// TIA Portal project "Paletizace trayů" (V14)

(* hardware
DEVICE "ET 200S station_1"  ET 200S station
   slot 0: "Rack_0"  Rail
   slot 2: "PLC_1"  IM 151-8 PN/DP CPU  6ES7 151-8AB01-0AB0  V3.2
      slot 1: "PROFINET interface_1"  PN-IO
         slot 1: "Port_1"  Port
         slot 2: "Port_2"  Port
         slot 3: "Port_3"  Port
   slot 4: "PM-E 24VDC_1"  PM-E 24VDC  6ES7 138-4CA01-0AA0
   slot 5: "4SI IO link_1"  4SI IO link  6ES7 138-4GA50-0AB0
   slot 6: "4SI IO link_2"  4SI IO link  6ES7 138-4GA50-0AB0
   slot 7: "4SI IO link_3"  4SI IO link  6ES7 138-4GA50-0AB0
   slot 8: "4SI IO link_4"  4SI IO link  6ES7 138-4GA50-0AB0
   slot 9: "PM-E 24VDC_2"  PM-E 24VDC  6ES7 138-4CA01-0AA0
   slot 10: "8DI x 24VDC_1"  8DI x 24VDC  6ES7 131-4BF00-0AA0
   slot 11: "8DI x 24VDC_2"  8DI x 24VDC  6ES7 131-4BF00-0AA0
   slot 12: "8DI x 24VDC_3"  8DI x 24VDC  6ES7 131-4BF00-0AA0
   slot 13: "8DI x 24VDC_4"  8DI x 24VDC  6ES7 131-4BF00-0AA0
   slot 14: "8DI x 24VDC_5"  8DI x 24VDC  6ES7 131-4BF00-0AA0
   slot 15: "8DI x 24VDC_6"  8DI x 24VDC  6ES7 131-4BF00-0AA0
   slot 16: "8DI x 24VDC_7"  8DI x 24VDC  6ES7 131-4BF00-0AA0
   slot 17: "8DI x 24VDC_8"  8DI x 24VDC  6ES7 131-4BF00-0AA0
   slot 18: "8DI x 24VDC_9"  8DI x 24VDC  6ES7 131-4BF00-0AA0
   slot 19: "8DI x 24VDC_10"  8DI x 24VDC  6ES7 131-4BF00-0AA0
   slot 20: "8DI x 24VDC_11"  8DI x 24VDC  6ES7 131-4BF00-0AA0
   slot 21: "8DI x 24VDC_12"  8DI x 24VDC  6ES7 131-4BF00-0AA0
   slot 22: "8DI x 24VDC_13"  8DI x 24VDC  6ES7 131-4BF00-0AA0
   slot 23: "8DI x 24VDC_14"  8DI x 24VDC  6ES7 131-4BF00-0AA0
   slot 24: "8DI x 24VDC_15"  8DI x 24VDC  6ES7 131-4BF00-0AA0
   slot 25: "8DI x 24VDC_16"  8DI x 24VDC  6ES7 131-4BF00-0AA0
   slot 26: "PM-E 24VDC_3"  PM-E 24VDC  6ES7 138-4CA01-0AA0
   slot 27: "8DO x 24VDC / 0.5A_1"  8DO x 24VDC / 0.5A  6ES7 132-4BF00-0AA0
   slot 28: "8DO x 24VDC / 0.5A_2"  8DO x 24VDC / 0.5A  6ES7 132-4BF00-0AA0
   slot 29: "PM-E 24VDC_4"  PM-E 24VDC  6ES7 138-4CA01-0AA0
   slot 30: "8DO x 24VDC / 0.5A_3"  8DO x 24VDC / 0.5A  6ES7 132-4BF00-0AA0
   slot 31: "8DO x 24VDC / 0.5A_4"  8DO x 24VDC / 0.5A  6ES7 132-4BF00-0AA0
   slot 32: "8DO x 24VDC / 0.5A_5"  8DO x 24VDC / 0.5A  6ES7 132-4BF00-0AA0
   slot 33: "8DO x 24VDC / 0.5A_6"  8DO x 24VDC / 0.5A  6ES7 132-4BF00-0AA0
   slot 34: "8DO x 24VDC / 0.5A_7"  8DO x 24VDC / 0.5A  6ES7 132-4BF00-0AA0
   slot 35: "8DO x 24VDC / 0.5A_8"  8DO x 24VDC / 0.5A  6ES7 132-4BF00-0AA0
   slot 36: "8DO x 24VDC / 0.5A_9"  8DO x 24VDC / 0.5A  6ES7 132-4BF00-0AA0
   slot 37: "8DO x 24VDC / 0.5A_10"  8DO x 24VDC / 0.5A  6ES7 132-4BF00-0AA0
   slot 38: "8DO x 24VDC / 0.5A_11"  8DO x 24VDC / 0.5A  6ES7 132-4BF00-0AA0
   slot 39: "PM-E 24VDC_5"  PM-E 24VDC  6ES7 138-4CA01-0AA0
   slot 40: "8DO x 24VDC / 0.5A_12"  8DO x 24VDC / 0.5A  6ES7 132-4BF00-0AA0
   slot 41: "8DO x 24VDC / 0.5A_13"  8DO x 24VDC / 0.5A  6ES7 132-4BF00-0AA0
   slot 42: "8DO x 24VDC / 0.5A_14"  8DO x 24VDC / 0.5A  6ES7 132-4BF00-0AA0
   slot 43: "8DO x 24VDC / 0.5A_15"  8DO x 24VDC / 0.5A  6ES7 132-4BF00-0AA0
   slot 44: "8DO x 24VDC / 0.5A_16"  8DO x 24VDC / 0.5A  6ES7 132-4BF00-0AA0
   slot 45: "8DO x 24VDC / 0.5A_17"  8DO x 24VDC / 0.5A  6ES7 132-4BF00-0AA0
   slot 46: "8DO x 24VDC / 0.5A_18"  8DO x 24VDC / 0.5A  6ES7 132-4BF00-0AA0
   slot 47: "8DO x 24VDC / 0.5A_19"  8DO x 24VDC / 0.5A  6ES7 132-4BF00-0AA0
   slot 48: "8DO x 24VDC / 0.5A_20"  8DO x 24VDC / 0.5A  6ES7 132-4BF00-0AA0
DEVICE "GSD device_1"  GSD.Device.PN
   slot 0: "Rack"  Rack  V1.0
   slot 0: "ComauR1"  X20IF10E3-1  X20IF10E3-1  2.1.x
      slot 0: "DIM 1"  DIM 1
      slot 1: "Interface"  Interface
         slot 1: "Interface - Port1"  Interface - Port1
         slot 2: "Interface - Port2"  Interface - Port2
   slot 1: "32 Bytes In_1"  32 Bytes In
      slot 0: "17"  17
   slot 2: "32 Bytes Out_1"  32 Bytes Out
      slot 0: "18"  18
DEVICE "GSD device_2"  GSD.Device.PN
   slot 0: "Rack"  Rack  V1.0
   slot 0: "ComauR2"  X20IF10E3-1  X20IF10E3-1  2.1.x
      slot 0: "DIM 1"  DIM 1
      slot 1: "Interface"  Interface
         slot 1: "Interface - Port1"  Interface - Port1
         slot 2: "Interface - Port2"  Interface - Port2
   slot 1: "32 Bytes In_1"  32 Bytes In
      slot 0: "17"  17
   slot 2: "32 Bytes Out_1"  32 Bytes Out
      slot 0: "18"  18
DEVICE "Panel paletizace trayů"  KTP600 Basic color PN
   slot 0: "KTP600 Basic color PN"  KTP600 Basic color PN  6AV6 647-0AD11-3AX0  12.0.0.0
   slot 1: "HMI_RT_2"  KTP600 Basic color PN  6AV6 647-0AD11-3AX0  12.0.0.0
   slot 5: "Panel paletizace trayů.IE_CP_1"  PROFINET Interface  12.0.0.0
      slot 1: "PROFINET Interface_1"  PROFINET Interface
         slot 1: "Port_1"  Port
DEVICE "GSD device_3"  GSD.Device.PN
   slot 0: "Rack"  Rack  V1.0
   slot 1: "rpt1ezp810-8"  plcEZP810-8  6ES7 214-1AG40-0XB0  V4.1
      slot 0: "MasterQ"  MasterQ
      slot 1: "MasterI"  MasterI
      slot 2: "Interface"  Interface
         slot 1: "Port 1"  Port 1
*)

// ===== PLC "PLC_1"  IM 151-8 PN/DP CPU =====

VAR_GLOBAL   // PLC tag table "Default tag table"
   "P12 nahoře" AT %I44.0 : Bool;
   "Zdvih P12B Nahoru" AT %Q17.6 : Bool;
   "Zdvih P12B Brzda" AT %Q18.0 : Bool;
   "Tag_5" AT %M2.0 : Bool;
   "P12 dole" AT %I44.1 : Bool;
   "Zdvih P11B Nahoru" AT %Q17.1 : Bool;
   "Zdvih P12B Dolu" AT %Q17.7 : Bool;
   "Tag_10" AT %Q33.0 : Bool;
   "Tlačítko zapnout" AT %I13.0 : Bool;
   "Tlačítko reset" AT %I13.1 : Bool;
   "Tag_13" AT %Q26.0 : Bool;
   "Tag_14" AT %Q26.1 : Bool;
   "Tag_15" AT %Q26.2 : Bool;
   "FM P35 Start" AT %Q20.3 : Bool;
   "Tag_17" AT %M4.0 : Bool;
   "Reset frekvenčních měničů" AT %Q25.5 : Bool;
   "Tag_19" AT %M4.1 : Bool;
   "Tlačítko override" AT %I13.2 : Bool;
   "Tag_21" AT %M5.0 : Bool;
   "FM P35 rychlost bit 0" AT %Q20.5 : Bool;
   "Tag_12" AT %M6.0 : Bool;
   "FM P35 rychlost bit 1" AT %Q20.6 : Bool;
   "Tag_16" AT %M9.0 : Bool;
   "FM P27 start" AT %Q19.4 : Bool;
   "Tag_20" AT %M4.2 : Bool;
   "Tag_22" AT %M60.0 : Bool;
   "Destohovač P6 nahoru" AT %Q16.3 : Bool;
   "Tag_23" AT %M60.1 : Bool;
   "Destohovač P6 dolu" AT %Q16.4 : Bool;
   "Destohovač P6 brzda" AT %Q16.5 : Bool;
   "Destohovač D6 Nahoře" AT %I40.5 : Bool;
   "Destohovač D6 Dole" AT %I40.7 : Bool;
   "Tag_26" AT %M1.4 : Bool;
   "Dopravník P4 Start" AT %Q16.1 : Bool;
   "Dopravník P5 Stohovač Start" AT %Q16.2 : Bool;
   "Tag_27" AT %M80.1 : Bool;
   "Tag_28" AT %M80.2 : Bool;
   "Dopravník P8 Start" AT %Q16.6 : Bool;
   "Tag_4" AT %M80.4 : Bool;
   "Tag_3" AT %M80.5 : Bool;
   "Dopravník 12 A start" AT %Q17.4 : Bool;
   "Tag_29" AT %M80.6 : Bool;
   "Dopravník 12 A vzad" AT %Q17.5 : Bool;
   "Tag_9" AT %M91.0 : Bool;
   "Dopravník P17 Start" AT %Q18.1 : Bool;
   "Dopravník P18 Start" AT %Q18.2 : Bool;
   "Dopravník Ovinovačka P19 start" AT %Q18.3 : Bool;
   "Tag_30" AT %M91.1 : Bool;
   "Tag_31" AT %M91.2 : Bool;
   "Tag_32" AT %M91.3 : Bool;
   "Dopravník P20 Start" AT %Q18.4 : Bool;
   "Tag_33" AT %M20.0 : Bool;
   "Tag_34" AT %M20.1 : Bool;
   "Zdvih P11B Dolu" AT %Q17.2 : Bool;
   "Zdvih P11B Brzda" AT %Q17.3 : Bool;
   "P11 dole" AT %I42.7 : Bool;
   "P11 nahoře" AT %I42.6 : Bool;
   "Tag_8" AT %M20.2 : Bool;
   "Dopravník P11A start" AT %Q16.7 : Bool;
   "Dopravník P11A vzad" AT %Q17.0 : Bool;
   "Tag_39" AT %M20.4 : Bool;
   "Tag_35" AT %M110.0 : Bool;
   "Dopravník P36 start" AT %Q20.7 : Bool;
   "Dopravník P37 Start" AT %Q21.0 : Bool;
   "Tag_36" AT %M110.1 : Bool;
   "FM P23.1 Start" AT %Q186.1 : Bool;
   "FM P23.2 Start" AT %Q19.1 : Bool;
   "FM P28 Start" AT %Q20.0 : Bool;
   "FM P29 Start" AT %Q20.1 : Bool;
   "P33 Start" AT %Q20.2 : Bool;
   "Tag_18" AT %Q19.6 : Bool;
   "Tag_40" AT %Q19.7 : Bool;
   "P 47.1 Start" AT %Q21.2 : Bool;
   "P 47.2 Start" AT %Q21.3 : Bool;
   "P 49 Start" AT %Q21.4 : Bool;
   "Rovnání palety P12 sevřít" AT %Q47.5 : Bool;
   "Rovnání palety P12 rozevřít" AT %Q47.4 : Bool;
   "Rovnání palety P11 sevřít" AT %Q47.1 : Bool;
   "Rovnání palety P11 rozevřít" AT %Q47.0 : Bool;
   "Destohovač sevřít" AT %Q41.7 : Bool;
   "Destohovač rozevřít" AT %Q41.6 : Bool;
   "Klapka 47.2 nahoru" AT %Q46.2 : Bool;
   "Klapka 47.2 dolů" AT %Q46.3 : Bool;
   "Klapka P47.1 nahoru" AT %Q46.0 : Bool;
   "Klapka P47.1 dolů" AT %Q46.1 : Bool;
   "Klapka P33 nahoru" AT %Q46.4 : Bool;
   "Klapka P33 dolů" AT %Q46.5 : Bool;
   "Paleta na konci P5" AT %I41.4 : Bool;
   "Destohovač D6 rameno pravé sevřeno" AT %I41.3 : Bool;
   "Paleta na P8 pozice 12" AT %I42.3 : Bool;
   "Tag_1" AT %I44.5 : Bool;
   "Paleta na P12" AT %I44.2 : Bool;
   "Tag_7" AT %Q47.2 : Bool;
   "PaletaNaD17pozice12" AT %I44.6 : Bool;
   "Tag_41" AT %T50 : Timer;
   "Paleta na konci P17" AT %I48.0 : Bool;
   "Tag_42" AT %T51 : Timer;
   "Spoždění ukončení automatu" AT %T0 : Timer;
   "Paleta na konci P18" AT %I48.1 : Bool;
   "Paleta v ovíječce P19" AT %I48.2 : Bool;
   "Paleta na Začátku P18" AT %I48.7 : Bool;
   "Paleta na Začátku P20" AT %I48.4 : Bool;
   "Paleta na konci P20" AT %I48.5 : Bool;
   "Karton na konci P47.2" AT %I55.1 : Bool;
   "Karton na začátku P49" AT %I59.1 : Bool;
   "Tag_43" AT %T40 : Timer;
   "Karton na konci P49" AT %I58.6 : Bool;
   "Konec řady na P49" AT %I58.7 : Bool;
   "Dojetá řada na P49" AT %I59.0 : Bool;
   "Karton na konci P47.1" AT %I55.2 : Bool;
   "Dopravník P47.2 plný" AT %I45.5 : Bool;
   "Tag_44" AT %M10.0 : Bool;
   "Tag_45" AT %M11.0 : Bool;
   "Tag_46" AT %M16.0 : Bool;
   "Tag_47" AT %M16.1 : Bool;
   "Tag_48" AT %T60 : Timer;
   "Tag_49" AT %T61 : Timer;
   "Tag_50" AT %T62 : Timer;
   "Tag_51" AT %T63 : Timer;
   "Silové obvody okruh 1 OK" AT %I14.0 : Bool;
   "Motorový jistič Destohovač D6 OK" AT %I0.1 : Bool;
   "Destohovač D6 havárie dole" AT %I0.7 : Bool;
   "Destohovač D6 havárie nahoře" AT %I0.6 : Bool;
   "Tlak vzduchu OK" AT %I3.7 : Bool;
   "Paleta pod destohovačem D6" AT %I40.4 : Bool;
   "Destohovač D6 Uprostřed" AT %I40.6 : Bool;
   "Destohovač D6 Rameno Levé otevřeno" AT %I41.0 : Bool;
   "Destohovač D6 rameno pravé otevřeno" AT %I41.2 : Bool;
   "Destohovač D6 rameno levé sevřeno" AT %I41.1 : Bool;
   "Tag_62" AT %I320.0 : Bool;
   "Tag_63" AT %M150.0 : Bool;
   "Tag_64" AT %M150.3 : Bool;
   "Tag_65" AT %Q320.0 : Bool;
   "Tag_66" AT %M100.0 : Bool;
   "Tag_67" AT %M100.1 : Bool;
   "Tag_68" AT %M120.0 : Bool;
   "Motorový jistič P3,P4,P5,P8 OK" AT %I0.0 : Bool;
   "Paleta na Začátku D8" AT %I45.6 : Bool;
   "Stoh palet na konci D4" AT %I40.2 : Bool;
   "Stoh palet na Začátku D5" AT %I40.3 : Bool;
   "Paleta na P8 pozice 11" AT %I42.2 : Bool;
   "Pomocná začátek přesunu na D12" AT %M61.1 : Bool;
   "Tag_24" AT %M120.1 : Bool;
   "Starttovací okno D18" AT %T52 : Timer;
   "Tag_25" AT %T41 : Timer;
   "Tag_37" AT %I54.7 : Bool;
   "Tag_38" AT %I54.3 : Bool;
   "Tag_52" AT %I54.1 : Bool;
   "Tag_53" AT %I54.4 : Bool;
   "Tag_54" AT %T42 : Timer;
   "Tag_55" AT %T44 : Timer;
   "Tag_56" AT %I54.2 : Bool;
   "Tag_57" AT %I54.0 : Bool;
   "Tag_58" AT %T45 : Timer;
   "Tag_59" AT %Q33.1 : Bool;
   "Tag_60" AT %Q33.3 : Bool;
   "Tag_70" AT %Q33.4 : Bool;
   "Tag_71" AT %Q33.5 : Bool;
   "Tag_72" AT %M2.1 : Bool;
   "Tag_73" AT %M2.2 : Bool;
   "Tag_2" AT %T2 : Timer;
   "Tag_6" AT %T90 : Timer;
   "Tag_11" AT %T91 : Timer;
END_VAR

VAR_GLOBAL   // PLC tag table "Tag table_1"
   "Ovíječka_Volná trať" AT %I10.0 : Bool;
   "Ovíječka_Konec balení" AT %I10.1 : Bool;
   "Ovíječka_Porucha" AT %I10.2 : Bool;
   "Ovíječka_Paleta na točně" AT %I10.3 : Bool;
   "Ovíječce_Start balení" AT %Q29.4 : Bool;
   "Ovíječce_Možno balit" AT %Q29.5 : Bool;
   "Tag_61" AT %Q29.6 : Bool;
   "Tag_69" AT %Q29.7 : Bool;
END_VAR

VAR_GLOBAL   // PLC tag table "System"
   "AlwaysTRUE" AT %M1.2 : Bool;
   "Clock memory bit 10 Hz" AT %M0.0 : Bool;
   "Clock memory bit 5 Hz" AT %M0.1 : Bool;
   "Clock memory bit 2.5 Hz" AT %M0.2 : Bool;
   "Clock memory bit 2 Hz" AT %M0.3 : Bool;
   "Clock memory bit 1.25 Hz" AT %M0.4 : Bool;
   "Clock memory bit 1 Hz" AT %M0.5 : Bool;
   "Clock memory bit 0.625 Hz" AT %M0.6 : Bool;
   "Clock memory bit 0.5 Hz" AT %M0.7 : Bool;
   "AlwaysFALSE" AT %M1.3 : Bool;
   "DiagStatusUpdate" AT %M1.1 : Bool;
   "FirstScan" AT %M1.0 : Bool;
END_VAR

TYPE "Artikl2"
   STRUCT
      Cislo : Int;
      Pocet : Int;
      Novy : Bool;
      Mlecny : Bool;
   END_STRUCT;
END_TYPE

TYPE "Artikl"
   STRUCT
      Novy : Bool;
      Mlecny : Bool;
      Mlecny4 : Bool;
      Mlecny6 : Bool;
      Mlecny8 : Bool;
      Mlecny9 : Bool;
      Mlecny99 : Bool;
      Mlecny9999 : Bool;
      Cislo : Word;
      Pocet : Word;
   END_STRUCT;
END_TYPE

TYPE "Pocet"
   STRUCT
      "Požadovaný počet vrstev" : Int;
      "Aktuální počet vrstev" : Int;
      "Aktuální počet půlvrstev" : Int;
   END_STRUCT;
END_TYPE

TYPE "Paleta"
   STRUCT
      Artik : String;
      "Počet vrstev" : Int;
      "Počet půlvrstev" : Int;
      "Neúplná paleta" : Bool;
   END_STRUCT;
END_TYPE

DATA_BLOCK "OB1"   // DB1
{ S7_Optimized_Access := 'FALSE' }
VERSION : 0.1
   VAR
      OB1_EV_CLASS : Byte;
      OB1_SCAN_1 : Byte;
      OB1_PRIORITY : Byte;
      OB1_OB_NUMBR : Byte;
      OB1_RESERVED_1 : Byte;
      OB1_RESERVED_2 : Byte;
      OB1_PREV_CYCLE : Int;
      OB1_MIN_CYCLE : Int;
      OB1_MAX_CYCLE : Int;
      OB1_DATE_TIME : Date_And_Time;
   END_VAR
BEGIN
END_DATA_BLOCK

DATA_BLOCK "Data_block_1"   // DB2
{ S7_Optimized_Access := 'FALSE' }
VERSION : 0.1
   VAR
      moje : Struct
         aa : Bool;
         aaaa : Bool;
      END_STRUCT;
      dd : Bool;
   END_VAR
BEGIN
END_DATA_BLOCK

DATA_BLOCK "Data_block_2"   // DB3
{ S7_Optimized_Access := 'FALSE' }
VERSION : 0.1
BEGIN
END_DATA_BLOCK

DATA_BLOCK "DataPole"   // DB4
{ S7_Optimized_Access := 'FALSE' }
VERSION : 0.1
   VAR
      Artikly : Array[0..100] of "Artikl2";
      Konci : Bool;
   END_VAR
BEGIN
END_DATA_BLOCK

DATA_BLOCK "Block_1_DB"   // DB5
{ S7_Optimized_Access := 'FALSE' }
VERSION : 0.1
// stored: InstanceOfName Block_1
"Block_1"
BEGIN
END_DATA_BLOCK

DATA_BLOCK "ArtiklDB"   // DB6
{ S7_Optimized_Access := 'FALSE' }
VERSION : 0.1
   VAR
      Artikl : "Artikl";
   END_VAR
BEGIN
END_DATA_BLOCK

DATA_BLOCK "Dopravníky palet_DB"   // DB8
{ S7_Optimized_Access := 'FALSE' }
VERSION : 0.1
// stored: InstanceOfName Dopravníky palet
"Dopravníky palet"
BEGIN
END_DATA_BLOCK

DATA_BLOCK "Data_block_3"   // DB9
{ S7_Optimized_Access := 'FALSE' }
VERSION : 0.1
   VAR
      artikl : Struct
         Novy : Bool;
         Mlecny : Bool;
         Mlecny4 : Bool;
         Mlecny6 : Bool;
         Mlecny8 : Bool;
         Mlecny9 : Bool;
         Mlecny99 : Bool;
         Mlecny9999 : Bool;
         Cislo : Word;
         Pocet : Word;
      END_STRUCT;
   END_VAR
BEGIN
END_DATA_BLOCK

DATA_BLOCK "Artikly"   // DB10
{ S7_Optimized_Access := 'FALSE' }
VERSION : 0.1
   VAR
      Artikly : Array[0..100] of "Artikl";
   END_VAR
BEGIN
END_DATA_BLOCK

DATA_BLOCK "Dopravníky kartonů linka 1_DB"   // DB11
{ S7_Optimized_Access := 'FALSE' }
VERSION : 0.1
// stored: InstanceOfName Dopravníky kartonů linka 1
"Dopravníky kartonů linka 1"
BEGIN
END_DATA_BLOCK

DATA_BLOCK "Globální řízení_DB"   // DB12
{ S7_Optimized_Access := 'FALSE' }
VERSION : 0.1
// stored: InstanceOfName Globální řízení
"Globální řízení"
BEGIN
END_DATA_BLOCK

DATA_BLOCK "Počítadlo_DB"   // DB15
{ S7_Optimized_Access := 'FALSE' }
VERSION : 0.1
// stored: InstanceOfName Počítadlo
"Počítadlo"
BEGIN
END_DATA_BLOCK

DATA_BLOCK "OPPovely"   // DB20
{ S7_Optimized_Access := 'FALSE' }
VERSION : 0.1
   VAR
      "OP Start" : Bool;
      "OP Stop" : Bool;
      "OP Manual" : Bool;
      "P3 Start" : Bool;
      "P4 Start" : Bool;
      "P5 Start" : Bool;
      "Destohovač nahoru" : Bool;
      "Destohovač dolu" : Bool;
      "Destohovač ramena sevřít" : Bool;
      "Destohovač ramena rozevřít" : Bool;
      "P8 Start" : Bool;
      "P12 Start" : Bool;
      "P12 Vzad" : Bool;
      "P12 Nahoru" : Bool;
      "P12 Dolu" : Bool;
      "P12 Rovnání" : Bool;
      "P11 Start" : Bool;
      "P11 Vzad" : Bool;
      "P11 Nahoru" : Bool;
      "P11 Dolu" : Bool;
      "P11 Rovnání" : Bool;
      "P17 Start" : Bool;
      "P18 Start" : Bool;
      "P19 Ovíječka Start" : Bool;
      "P20 Start" : Bool;
      "P21 Start" : Bool;
      Linka1 : Struct
         "P23 Start" : Bool;
         "P28 Start" : Bool;
         "P27 Elevátor Start" : Bool;
         "P29 Start" : Bool;
         "P33 Start" : Bool;
         "Klapka P33" : Bool;
         "P36 Start" : Bool;
         "P35 Elevátor Start" : Bool;
         "P37 Start" : Bool;
         "P47.1 Start" : Bool;
         "Klapka P47.1" : Bool;
         "P47.2 Start" : Bool;
         "Klapka P47.2" : Bool;
         "P49 Start" : Bool;
         reserve : Word;
      END_STRUCT;
   END_VAR
BEGIN
END_DATA_BLOCK

DATA_BLOCK "OPPovely Positivní Hrana"   // DB21
{ S7_Optimized_Access := 'FALSE' }
VERSION : 0.1
   VAR
      "OP Start" : Bool;
      "OP Stop" : Bool;
      "OP Manual" : Bool;
      "P3 Start" : Bool;
      "P4 Start" : Bool;
      "P5 Start" : Bool;
      "Destohovač nahoru" : Bool;
      "Destohovač dolu" : Bool;
      "Destohovač ramena sevřít" : Bool;
      "Destohovač ramena rozevřít" : Bool;
      "P8 Start" : Bool;
      "P12 Start" : Bool;
      "P12 Vzad" : Bool;
      "P12 Nahoru" : Bool;
      "P12 Dolu" : Bool;
      "P12 Rovnání" : Bool;
      "P11 Start" : Bool;
      "P11 Vzad" : Bool;
      "P11 Nahoru" : Bool;
      "P11 Dolu" : Bool;
      "P11 Rovnání" : Bool;
      "P17 Start" : Bool;
      "P18 Start" : Bool;
      "P19 Ovíječka Start" : Bool;
      "P20 Start" : Bool;
      "P21 Start" : Bool;
      Linka1 : Struct
         "P23 Start" : Bool;
         "P28 Start" : Bool;
         "P27 Elevátor Start" : Bool;
         "P29 Start" : Bool;
         "P33 Start" : Bool;
         "Klapka P33" : Bool;
         "P36 Start" : Bool;
         "P35 Elevátor Start" : Bool;
         "P37 Start" : Bool;
         "P47.1 Start" : Bool;
         "Klapka P47.1" : Bool;
         "P47.2 Start" : Bool;
         "Klapka P47.2" : Bool;
         "P49 Start" : Bool;
         reserve : Word;
      END_STRUCT;
   END_VAR
BEGIN
END_DATA_BLOCK

DATA_BLOCK "OPPovely Negativní Hrana"   // DB22
{ S7_Optimized_Access := 'FALSE' }
VERSION : 0.1
   VAR
      "OP Start" : Bool;
      "OP Stop" : Bool;
      "OP Manual" : Bool;
      "P3 Start" : Bool;
      "P4 Start" : Bool;
      "P5 Start" : Bool;
      "Destohovač nahoru" : Bool;
      "Destohovač dolu" : Bool;
      "Destohovač ramena sevřít" : Bool;
      "Destohovač ramena rozevřít" : Bool;
      "P8 Start" : Bool;
      "P12 Start" : Bool;
      "P12 Vzad" : Bool;
      "P12 Nahoru" : Bool;
      "P12 Dolu" : Bool;
      "P12 Rovnání" : Bool;
      "P11 Start" : Bool;
      "P11 Vzad" : Bool;
      "P11 Nahoru" : Bool;
      "P11 Dolu" : Bool;
      "P11 Rovnání" : Bool;
      "P17 Start" : Bool;
      "P18 Start" : Bool;
      "P19 Ovíječka Start" : Bool;
      "P20 Start" : Bool;
      "P21 Start" : Bool;
      Linka1 : Struct
         "P23 Start" : Bool;
         "P28 Start" : Bool;
         "P27 Elevátor Start" : Bool;
         "P29 Start" : Bool;
         "P33 Start" : Bool;
         "Klapka P33" : Bool;
         "P36 Start" : Bool;
         "P35 Elevátor Start" : Bool;
         "P37 Start" : Bool;
         "P47.1 Start" : Bool;
         "Klapka P47.1" : Bool;
         "P47.2 Start" : Bool;
         "Klapka P47.2" : Bool;
         "P49 Start" : Bool;
         reserve : Word;
      END_STRUCT;
   END_VAR
BEGIN
END_DATA_BLOCK

FUNCTION_BLOCK "Block_1"   // FB1, LAD
{ S7_Optimized_Access := 'FALSE' }
VERSION : 0.1
BEGIN
END_FUNCTION_BLOCK

FUNCTION_BLOCK "Dopravníky palet"   // FB2, LAD
{ S7_Optimized_Access := 'FALSE' }
VERSION : 0.1
   VAR
      Přesun : Struct
         KonecD4naDestohovač : Bool;
         DestohovačNaKonecD5 : Bool;
         KonecD5naZačátekD8 : Bool;
         ZačátekD8naD8x12 : Bool;
         D8x12naD8x11 : Bool;
         D8x12naD12 : Bool;
         D8x11naD11 : Bool;
         D12naD17x12 : Bool;
         D11naD17x11 : Bool;
         D17x12naKonecP17 : Bool;
         D17x11naKonecP17 : Bool;
         KonecP17naZačátekP18 : Bool;
         ZačátekP18naKonecP18 : Bool;
         KonecP18naP19 : Bool;
         P19naZačátekP20 : Bool;
         ZačátekP20naKonecP20 : Bool;
         KonecP20NaP21 : Bool;
      END_STRUCT;
      "Přesun zahájen" : Struct
         KonecD4naDestohovač : Bool;
         DestohovačNaKonecD5 : Bool;
         KonecD5naZačátekD8 : Bool;
         ZačátekD8naD8x12 : Bool;
         D8x12naD8x11 : Bool;
         D8x12naD12 : Bool;
         D8x11naD11 : Bool;
         D12naD17x12 : Bool;
         D11naD17x11 : Bool;
         D17x12naKonecP17 : Bool;
         D17x11naKonecP17 : Bool;
         KonecP17naZačátekP18 : Bool;
         ZačátekP18naKonecP18 : Bool;
         KonecP18naP19 : Bool;
         P19naZačátekP20 : Bool;
         ZačátekP20naKonecP20 : Bool;
         KonecP20NaP21 : Bool;
      END_STRUCT;
      "Přesun zahájen paměť hrany" : Struct
         KonecD4naDestohovač : Bool;
         DestohovačNaKonecD5 : Bool;
         KonecD5naZačátekD8 : Bool;
         ZačátekD8naD8x12 : Bool;
         D8pozice12naD8x11 : Bool;
         D8x12naD12 : Bool;
         D8x11naD11 : Bool;
         D12naD17x12 : Bool;
         D11naD17x11 : Bool;
         D17x12naKonecP17 : Bool;
         D17x11naKonecP17 : Bool;
         KonecP17naZačátekP18 : Bool;
         ZačátekP18naKonecP18 : Bool;
         KonecP18naP19 : Bool;
         P19naZačátekP20 : Bool;
         ZačátekP20naKonecP20 : Bool;
         KonecP20NaP21 : Bool;
      END_STRUCT;
      "Přítomnosti palet" : Struct
         PaletaPodDestohovačem : Bool;
         PaletaNaKonciD5 : Bool;
         PaletaNaZačátkuD8 : Bool;
         PaletaNaD8pozice12 : Bool;
         PaletaNaD8pozice11 : Bool;
         PaletaNaP12 : Bool;
         PaletaNaP11 : Bool;
         PaletaNaD17pozice12 : Bool;
         PaletaNaD17pozice11 : Bool;
         PaletaNaKonciP17 : Bool;
         "PaletaNaZačátku P18" : Bool;
         PaletaNaKonciP18 : Bool;
         PaletaNaP19 : Bool;
         PaletaNaZačátkuP20 : Bool;
         PaletaNaKonciP20 : Bool;
      END_STRUCT;
      "Nájezdy palet" : Struct
         PaletaPodDestohovačem : Bool;
         PaletaNaKonciD5 : Bool;
         PaletaNaZačátkuD8 : Bool;
         PaletaNaD8pozice12 : Bool;
         PaletaNaD8pozice11 : Bool;
         PaletaNaP12 : Bool;
         PaletaNaP11 : Bool;
         PaletaNaD17pozice12 : Bool;
         PaletaNaD17pozice11 : Bool;
         PaletaNaKonciP17 : Bool;
         "PaletaNaZačátku P18" : Bool;
         PaletaNaKonciP18 : Bool;
         PaletaNaP19 : Bool;
         PaletaNaZačátkuP20 : Bool;
         PaletaNaKonciP20 : Bool;
      END_STRUCT;
      Palety : Struct
         P12 : "Paleta";
         P11 : "Paleta";
         P17poziceP11 : "Paleta";
         P17poziceP12 : "Paleta";
         KonecP17 : "Paleta";
         ZačátekP18 : "Paleta";
         KonecP18 : "Paleta";
         P19 : "Paleta";
         ZačátekP20 : "Paleta";
      END_STRUCT;
      Hrany : Struct
         T51Negativní : Bool;
      END_STRUCT;
      "Pallet dispenser_Instance" : "Pallet dispenser";
      "Přítomnost palety_Instance" : "Přítomnost palety";
   END_VAR
   VAR_TEMP
      Dummy : Bool;
      "Rovnání P11 sevřít" : Bool;
      "Rovnání P11 rozevřít" : Bool;
      "Rovnání P12 sevřít" : Bool;
      "Rovnání P12 rozevřít" : Bool;
      "Destohovač sevřít" : Bool;
      "Destohovač rozevřít" : Bool;
      "D12 Nahoru" : Bool;
   END_VAR
   VAR_TEMP   // added for the SCL form of the ladder/FBD networks
      _s5time1 : S5Time;
      _w1 : Bool;
      _w2 : Bool;
      _w3 : Bool;
   END_VAR
BEGIN

REGION Network 1
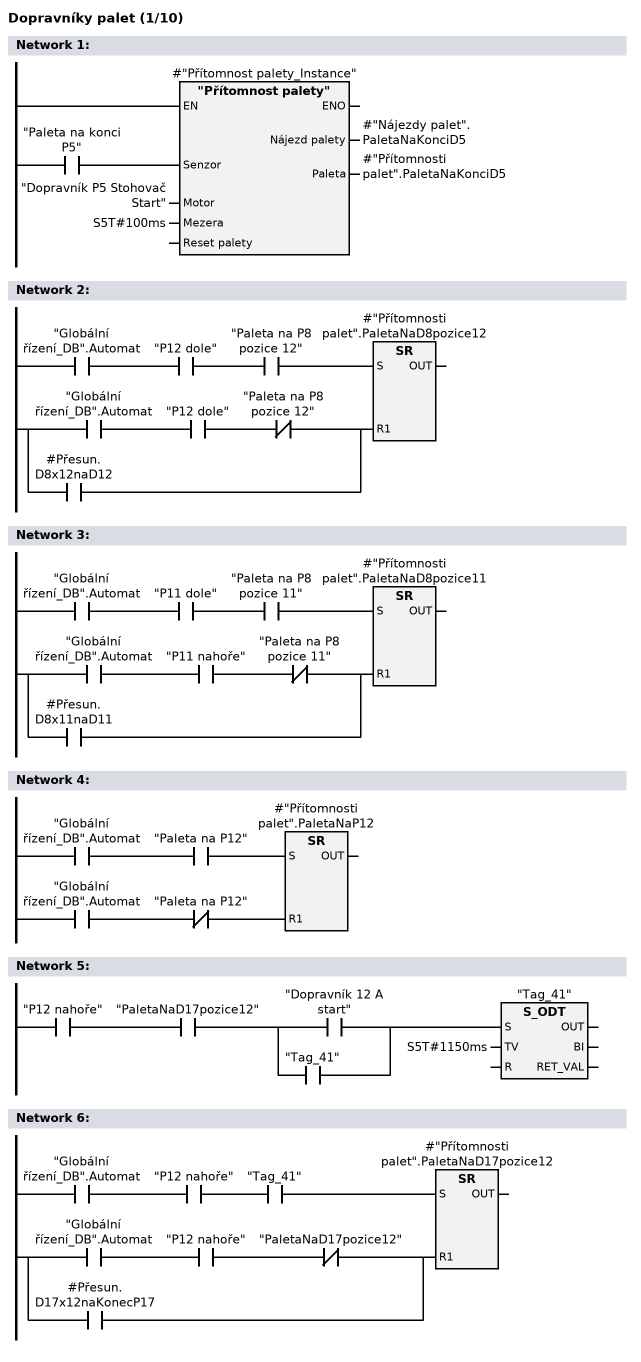
   RUNG wire#powerrail
      #"Přítomnost palety_Instance"(Senzor := wire#w1, Motor := "Dopravník P5 Stohovač Start", Mezera := S5T#100ms, "Reset palety" :=, "Nájezd palety" => #"Nájezdy palet".PaletaNaKonciD5, Paleta => #"Přítomnosti palet".PaletaNaKonciD5)
   END_RUNG
   RUNG wire#powerrail
      Contact( "Paleta na konci P5" )
   END_RUNG wire#w1
   // the same network as SCL:
   #"Přítomnost palety_Instance"(Senzor := "Paleta na konci P5",   // "Přítomnost palety"
                           Motor := "Dopravník P5 Stohovač Start",
                           Mezera := S5T#100ms,
                           "Nájezd palety" => #"Nájezdy palet".PaletaNaKonciD5,
                           Paleta => #"Přítomnosti palet".PaletaNaKonciD5);
END_REGION

REGION Network 2
   RUNG wire#powerrail
      Contact( "Globální řízení_DB".Automat )
      Contact( "P12 dole" )
      Contact( "Paleta na P8 pozice 12" )
      S_SR(operand := #"Přítomnosti palet".PaletaNaD8pozice12, r1 := wire#w1)
   END_RUNG
   RUNG wire#powerrail
      Contact( "Globální řízení_DB".Automat )
      Contact( "P12 dole" )
      I_Contact( "Paleta na P8 pozice 12" )
   END_RUNG wire#w1
   RUNG wire#powerrail
      Contact( #Přesun.D8x12naD12 )
   END_RUNG wire#w1
   // the same network as SCL:
   IF "Globální řízení_DB".Automat AND "P12 dole" AND "Paleta na P8 pozice 12" THEN
       #"Přítomnosti palet".PaletaNaD8pozice12 := TRUE;   // SR flip-flop
   END_IF;
   IF ("Globální řízení_DB".Automat AND "P12 dole" AND NOT "Paleta na P8 pozice 12") OR #Přesun.D8x12naD12 THEN
       #"Přítomnosti palet".PaletaNaD8pozice12 := FALSE;
   END_IF;
END_REGION

REGION Network 3
   RUNG wire#powerrail
      Contact( "Globální řízení_DB".Automat )
      Contact( "P11 dole" )
      Contact( "Paleta na P8 pozice 11" )
      S_SR(operand := #"Přítomnosti palet".PaletaNaD8pozice11, r1 := wire#w1)
   END_RUNG
   RUNG wire#powerrail
      Contact( "Globální řízení_DB".Automat )
      Contact( "P11 nahoře" )
      I_Contact( "Paleta na P8 pozice 11" )
   END_RUNG wire#w1
   RUNG wire#powerrail
      Contact( #Přesun.D8x11naD11 )
   END_RUNG wire#w1
   // the same network as SCL:
   IF "Globální řízení_DB".Automat AND "P11 dole" AND "Paleta na P8 pozice 11" THEN
       #"Přítomnosti palet".PaletaNaD8pozice11 := TRUE;   // SR flip-flop
   END_IF;
   IF ("Globální řízení_DB".Automat AND "P11 nahoře" AND NOT "Paleta na P8 pozice 11") OR #Přesun.D8x11naD11 THEN
       #"Přítomnosti palet".PaletaNaD8pozice11 := FALSE;
   END_IF;
END_REGION

REGION Network 4
   RUNG wire#powerrail
      Contact( "Globální řízení_DB".Automat )
      Contact( "Paleta na P12" )
      S_SR(operand := #"Přítomnosti palet".PaletaNaP12, r1 := wire#w1)
   END_RUNG
   RUNG wire#powerrail
      Contact( "Globální řízení_DB".Automat )
      I_Contact( "Paleta na P12" )
   END_RUNG wire#w1
   // the same network as SCL:
   IF "Globální řízení_DB".Automat AND "Paleta na P12" THEN
       #"Přítomnosti palet".PaletaNaP12 := TRUE;   // SR flip-flop
   END_IF;
   IF "Globální řízení_DB".Automat AND NOT "Paleta na P12" THEN
       #"Přítomnosti palet".PaletaNaP12 := FALSE;
   END_IF;
END_REGION

REGION Network 5
   RUNG wire#powerrail
      Contact( "P12 nahoře" )
      Contact( "PaletaNaD17pozice12" )
      wire#w1
      Contact( "Dopravník 12 A start" )
      wire#w2
      S_ODT(T_NO := "Tag_41", TV := S5T#1150ms, R :=, BI =>, RET_VAL =>)
   END_RUNG
   RUNG wire#w1
      Contact( "Tag_41" )
   END_RUNG wire#w2
   // the same network as SCL:
   #_s5time1 := S_ODT(T_NO := "Tag_41",
                      S := "P12 nahoře" AND "PaletaNaD17pozice12" AND ("Dopravník 12 A start" OR "Tag_41"),
                      TV := S5T#1150ms);
END_REGION

REGION Network 6
   RUNG wire#powerrail
      Contact( "Globální řízení_DB".Automat )
      Contact( "P12 nahoře" )
      Contact( "Tag_41" )
      S_SR(operand := #"Přítomnosti palet".PaletaNaD17pozice12, r1 := wire#w1)
   END_RUNG
   RUNG wire#powerrail
      Contact( "Globální řízení_DB".Automat )
      Contact( "P12 nahoře" )
      I_Contact( "PaletaNaD17pozice12" )
   END_RUNG wire#w1
   RUNG wire#powerrail
      Contact( #Přesun.D17x12naKonecP17 )
   END_RUNG wire#w1
   // the same network as SCL:
   IF "Globální řízení_DB".Automat AND "P12 nahoře" AND "Tag_41" THEN
       #"Přítomnosti palet".PaletaNaD17pozice12 := TRUE;   // SR flip-flop
   END_IF;
   IF ("Globální řízení_DB".Automat AND "P12 nahoře" AND NOT "PaletaNaD17pozice12") OR #Přesun.D17x12naKonecP17 THEN
       #"Přítomnosti palet".PaletaNaD17pozice12 := FALSE;
   END_IF;
END_REGION

REGION Network 7
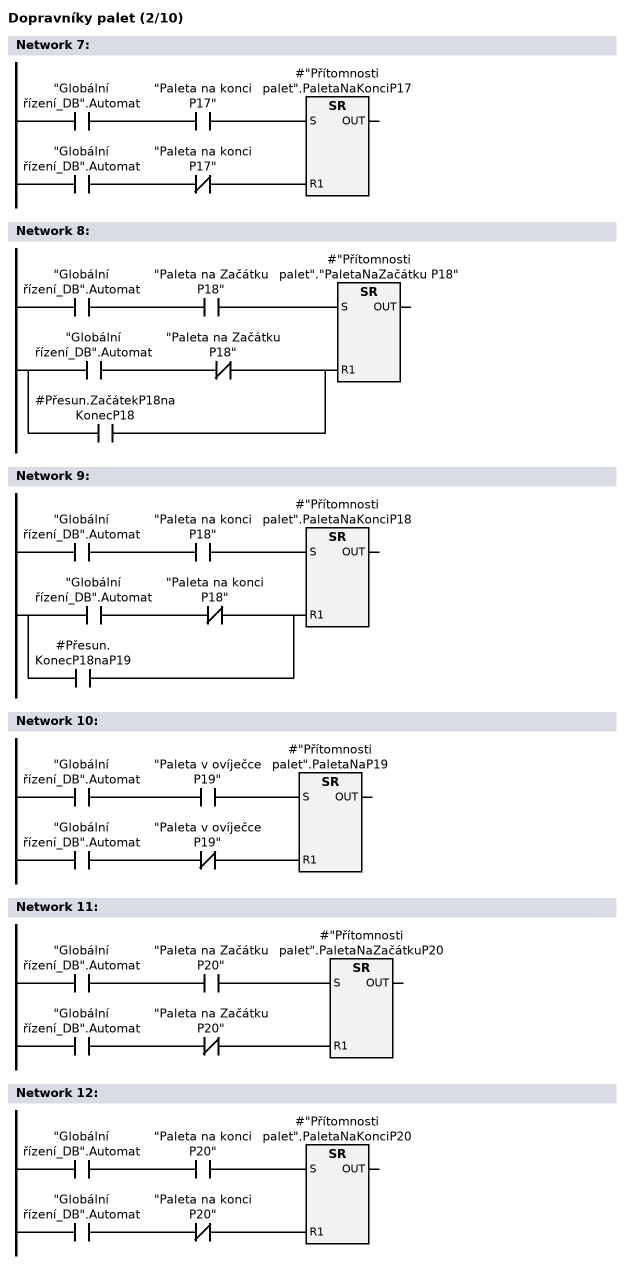
   RUNG wire#powerrail
      Contact( "Globální řízení_DB".Automat )
      Contact( "Paleta na konci P17" )
      S_SR(operand := #"Přítomnosti palet".PaletaNaKonciP17, r1 := wire#w1)
   END_RUNG
   RUNG wire#powerrail
      Contact( "Globální řízení_DB".Automat )
      I_Contact( "Paleta na konci P17" )
   END_RUNG wire#w1
   // the same network as SCL:
   IF "Globální řízení_DB".Automat AND "Paleta na konci P17" THEN
       #"Přítomnosti palet".PaletaNaKonciP17 := TRUE;   // SR flip-flop
   END_IF;
   IF "Globální řízení_DB".Automat AND NOT "Paleta na konci P17" THEN
       #"Přítomnosti palet".PaletaNaKonciP17 := FALSE;
   END_IF;
END_REGION

REGION Network 8
   RUNG wire#powerrail
      Contact( "Globální řízení_DB".Automat )
      Contact( "Paleta na Začátku P18" )
      S_SR(operand := #"Přítomnosti palet"."PaletaNaZačátku P18", r1 := wire#w1)
   END_RUNG
   RUNG wire#powerrail
      Contact( "Globální řízení_DB".Automat )
      I_Contact( "Paleta na Začátku P18" )
   END_RUNG wire#w1
   RUNG wire#powerrail
      Contact( #Přesun.ZačátekP18naKonecP18 )
   END_RUNG wire#w1
   // the same network as SCL:
   IF "Globální řízení_DB".Automat AND "Paleta na Začátku P18" THEN
       #"Přítomnosti palet"."PaletaNaZačátku P18" := TRUE;   // SR flip-flop
   END_IF;
   IF ("Globální řízení_DB".Automat AND NOT "Paleta na Začátku P18") OR #Přesun.ZačátekP18naKonecP18 THEN
       #"Přítomnosti palet"."PaletaNaZačátku P18" := FALSE;
   END_IF;
END_REGION

REGION Network 9
   RUNG wire#powerrail
      Contact( "Globální řízení_DB".Automat )
      Contact( "Paleta na konci P18" )
      S_SR(operand := #"Přítomnosti palet".PaletaNaKonciP18, r1 := wire#w1)
   END_RUNG
   RUNG wire#powerrail
      Contact( "Globální řízení_DB".Automat )
      I_Contact( "Paleta na konci P18" )
   END_RUNG wire#w1
   RUNG wire#powerrail
      Contact( #Přesun.KonecP18naP19 )
   END_RUNG wire#w1
   // the same network as SCL:
   IF "Globální řízení_DB".Automat AND "Paleta na konci P18" THEN
       #"Přítomnosti palet".PaletaNaKonciP18 := TRUE;   // SR flip-flop
   END_IF;
   IF ("Globální řízení_DB".Automat AND NOT "Paleta na konci P18") OR #Přesun.KonecP18naP19 THEN
       #"Přítomnosti palet".PaletaNaKonciP18 := FALSE;
   END_IF;
END_REGION

REGION Network 10
   RUNG wire#powerrail
      Contact( "Globální řízení_DB".Automat )
      Contact( "Paleta v ovíječce P19" )
      S_SR(operand := #"Přítomnosti palet".PaletaNaP19, r1 := wire#w1)
   END_RUNG
   RUNG wire#powerrail
      Contact( "Globální řízení_DB".Automat )
      I_Contact( "Paleta v ovíječce P19" )
   END_RUNG wire#w1
   // the same network as SCL:
   IF "Globální řízení_DB".Automat AND "Paleta v ovíječce P19" THEN
       #"Přítomnosti palet".PaletaNaP19 := TRUE;   // SR flip-flop
   END_IF;
   IF "Globální řízení_DB".Automat AND NOT "Paleta v ovíječce P19" THEN
       #"Přítomnosti palet".PaletaNaP19 := FALSE;
   END_IF;
END_REGION

REGION Network 11
   RUNG wire#powerrail
      Contact( "Globální řízení_DB".Automat )
      Contact( "Paleta na Začátku P20" )
      S_SR(operand := #"Přítomnosti palet".PaletaNaZačátkuP20, r1 := wire#w1)
   END_RUNG
   RUNG wire#powerrail
      Contact( "Globální řízení_DB".Automat )
      I_Contact( "Paleta na Začátku P20" )
   END_RUNG wire#w1
   // the same network as SCL:
   IF "Globální řízení_DB".Automat AND "Paleta na Začátku P20" THEN
       #"Přítomnosti palet".PaletaNaZačátkuP20 := TRUE;   // SR flip-flop
   END_IF;
   IF "Globální řízení_DB".Automat AND NOT "Paleta na Začátku P20" THEN
       #"Přítomnosti palet".PaletaNaZačátkuP20 := FALSE;
   END_IF;
END_REGION

REGION Network 12
   RUNG wire#powerrail
      Contact( "Globální řízení_DB".Automat )
      Contact( "Paleta na konci P20" )
      S_SR(operand := #"Přítomnosti palet".PaletaNaKonciP20, r1 := wire#w1)
   END_RUNG
   RUNG wire#powerrail
      Contact( "Globální řízení_DB".Automat )
      I_Contact( "Paleta na konci P20" )
   END_RUNG wire#w1
   // the same network as SCL:
   IF "Globální řízení_DB".Automat AND "Paleta na konci P20" THEN
       #"Přítomnosti palet".PaletaNaKonciP20 := TRUE;   // SR flip-flop
   END_IF;
   IF "Globální řízení_DB".Automat AND NOT "Paleta na konci P20" THEN
       #"Přítomnosti palet".PaletaNaKonciP20 := FALSE;
   END_IF;
END_REGION

REGION Network 13
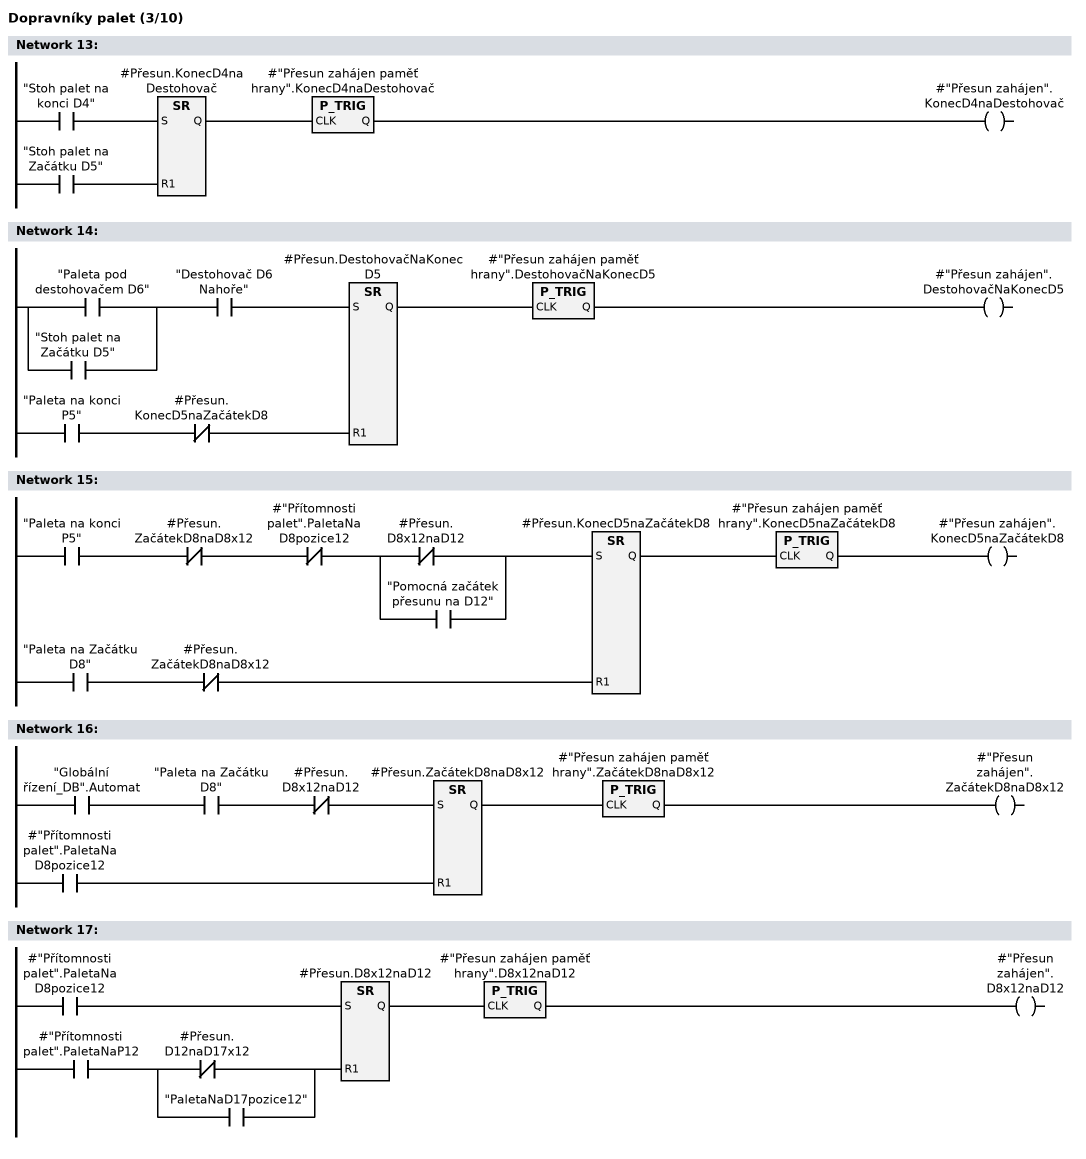
   RUNG wire#powerrail
      Contact( "Stoh palet na konci D4" )
      S_SR(operand := #Přesun.KonecD4naDestohovač, r1 := wire#w1)
      P_Trig( #"Přesun zahájen paměť hrany".KonecD4naDestohovač )
      Coil( #"Přesun zahájen".KonecD4naDestohovač )
   END_RUNG
   RUNG wire#powerrail
      Contact( "Stoh palet na Začátku D5" )
   END_RUNG wire#w1
   // the same network as SCL:
   IF "Stoh palet na konci D4" THEN
       #Přesun.KonecD4naDestohovač := TRUE;   // SR flip-flop
   END_IF;
   IF "Stoh palet na Začátku D5" THEN #Přesun.KonecD4naDestohovač := FALSE; END_IF;
   #_w1 := #Přesun.KonecD4naDestohovač AND NOT #"Přesun zahájen paměť hrany".KonecD4naDestohovač;   // rising edge
   #"Přesun zahájen paměť hrany".KonecD4naDestohovač := #Přesun.KonecD4naDestohovač;
   #"Přesun zahájen".KonecD4naDestohovač := #_w1;
END_REGION

REGION Network 14
   RUNG wire#powerrail
      Contact( "Paleta pod destohovačem D6" )
      wire#w1
      Contact( "Destohovač D6 Nahoře" )
      S_SR(operand := #Přesun.DestohovačNaKonecD5, r1 := wire#w2)
      P_Trig( #"Přesun zahájen paměť hrany".DestohovačNaKonecD5 )
      Coil( #"Přesun zahájen".DestohovačNaKonecD5 )
   END_RUNG
   RUNG wire#powerrail
      Contact( "Stoh palet na Začátku D5" )
   END_RUNG wire#w1
   RUNG wire#powerrail
      Contact( "Paleta na konci P5" )
      I_Contact( #Přesun.KonecD5naZačátekD8 )
   END_RUNG wire#w2
   // the same network as SCL:
   IF ("Paleta pod destohovačem D6" OR "Stoh palet na Začátku D5") AND "Destohovač D6 Nahoře" THEN
       #Přesun.DestohovačNaKonecD5 := TRUE;   // SR flip-flop
   END_IF;
   IF "Paleta na konci P5" AND NOT #Přesun.KonecD5naZačátekD8 THEN
       #Přesun.DestohovačNaKonecD5 := FALSE;
   END_IF;
   #_w1 := #Přesun.DestohovačNaKonecD5 AND NOT #"Přesun zahájen paměť hrany".DestohovačNaKonecD5;   // rising edge
   #"Přesun zahájen paměť hrany".DestohovačNaKonecD5 := #Přesun.DestohovačNaKonecD5;
   #"Přesun zahájen".DestohovačNaKonecD5 := #_w1;
END_REGION

REGION Network 15
   RUNG wire#powerrail
      Contact( "Paleta na konci P5" )
      I_Contact( #Přesun.ZačátekD8naD8x12 )
      I_Contact( #"Přítomnosti palet".PaletaNaD8pozice12 )
      wire#w1
      I_Contact( #Přesun.D8x12naD12 )
      wire#w2
      S_SR(operand := #Přesun.KonecD5naZačátekD8, r1 := wire#w3)
      P_Trig( #"Přesun zahájen paměť hrany".KonecD5naZačátekD8 )
      Coil( #"Přesun zahájen".KonecD5naZačátekD8 )
   END_RUNG
   RUNG wire#w1
      Contact( "Pomocná začátek přesunu na D12" )
   END_RUNG wire#w2
   RUNG wire#powerrail
      Contact( "Paleta na Začátku D8" )
      I_Contact( #Přesun.ZačátekD8naD8x12 )
   END_RUNG wire#w3
   // the same network as SCL:
   IF "Paleta na konci P5" AND NOT #Přesun.ZačátekD8naD8x12 AND NOT #"Přítomnosti palet".PaletaNaD8pozice12 AND (NOT #Přesun.D8x12naD12 OR "Pomocná začátek přesunu na D12") THEN
       #Přesun.KonecD5naZačátekD8 := TRUE;   // SR flip-flop
   END_IF;
   IF "Paleta na Začátku D8" AND NOT #Přesun.ZačátekD8naD8x12 THEN
       #Přesun.KonecD5naZačátekD8 := FALSE;
   END_IF;
   #_w1 := #Přesun.KonecD5naZačátekD8 AND NOT #"Přesun zahájen paměť hrany".KonecD5naZačátekD8;   // rising edge
   #"Přesun zahájen paměť hrany".KonecD5naZačátekD8 := #Přesun.KonecD5naZačátekD8;
   #"Přesun zahájen".KonecD5naZačátekD8 := #_w1;
END_REGION

REGION Network 16
   RUNG wire#powerrail
      Contact( "Globální řízení_DB".Automat )
      Contact( "Paleta na Začátku D8" )
      I_Contact( #Přesun.D8x12naD12 )
      S_SR(operand := #Přesun.ZačátekD8naD8x12, r1 := wire#w1)
      P_Trig( #"Přesun zahájen paměť hrany".ZačátekD8naD8x12 )
      Coil( #"Přesun zahájen".ZačátekD8naD8x12 )
   END_RUNG
   RUNG wire#powerrail
      Contact( #"Přítomnosti palet".PaletaNaD8pozice12 )
   END_RUNG wire#w1
   // the same network as SCL:
   IF "Globální řízení_DB".Automat AND "Paleta na Začátku D8" AND NOT #Přesun.D8x12naD12 THEN
       #Přesun.ZačátekD8naD8x12 := TRUE;   // SR flip-flop
   END_IF;
   IF #"Přítomnosti palet".PaletaNaD8pozice12 THEN #Přesun.ZačátekD8naD8x12 := FALSE; END_IF;
   #_w1 := #Přesun.ZačátekD8naD8x12 AND NOT #"Přesun zahájen paměť hrany".ZačátekD8naD8x12;   // rising edge
   #"Přesun zahájen paměť hrany".ZačátekD8naD8x12 := #Přesun.ZačátekD8naD8x12;
   #"Přesun zahájen".ZačátekD8naD8x12 := #_w1;
END_REGION

REGION Network 17
   RUNG wire#powerrail
      Contact( #"Přítomnosti palet".PaletaNaD8pozice12 )
      S_SR(operand := #Přesun.D8x12naD12, r1 := wire#w2)
      P_Trig( #"Přesun zahájen paměť hrany".D8x12naD12 )
      Coil( #"Přesun zahájen".D8x12naD12 )
   END_RUNG
   RUNG wire#powerrail
      Contact( #"Přítomnosti palet".PaletaNaP12 )
      wire#w1
      I_Contact( #Přesun.D12naD17x12 )
   END_RUNG wire#w2
   RUNG wire#w1
      Contact( "PaletaNaD17pozice12" )
   END_RUNG wire#w2
   // the same network as SCL:
   IF #"Přítomnosti palet".PaletaNaD8pozice12 THEN
       #Přesun.D8x12naD12 := TRUE;   // SR flip-flop
   END_IF;
   IF #"Přítomnosti palet".PaletaNaP12 AND (NOT #Přesun.D12naD17x12 OR "PaletaNaD17pozice12") THEN
       #Přesun.D8x12naD12 := FALSE;
   END_IF;
   #_w1 := #Přesun.D8x12naD12 AND NOT #"Přesun zahájen paměť hrany".D8x12naD12;   // rising edge
   #"Přesun zahájen paměť hrany".D8x12naD12 := #Přesun.D8x12naD12;
   #"Přesun zahájen".D8x12naD12 := #_w1;
END_REGION

REGION Network 18
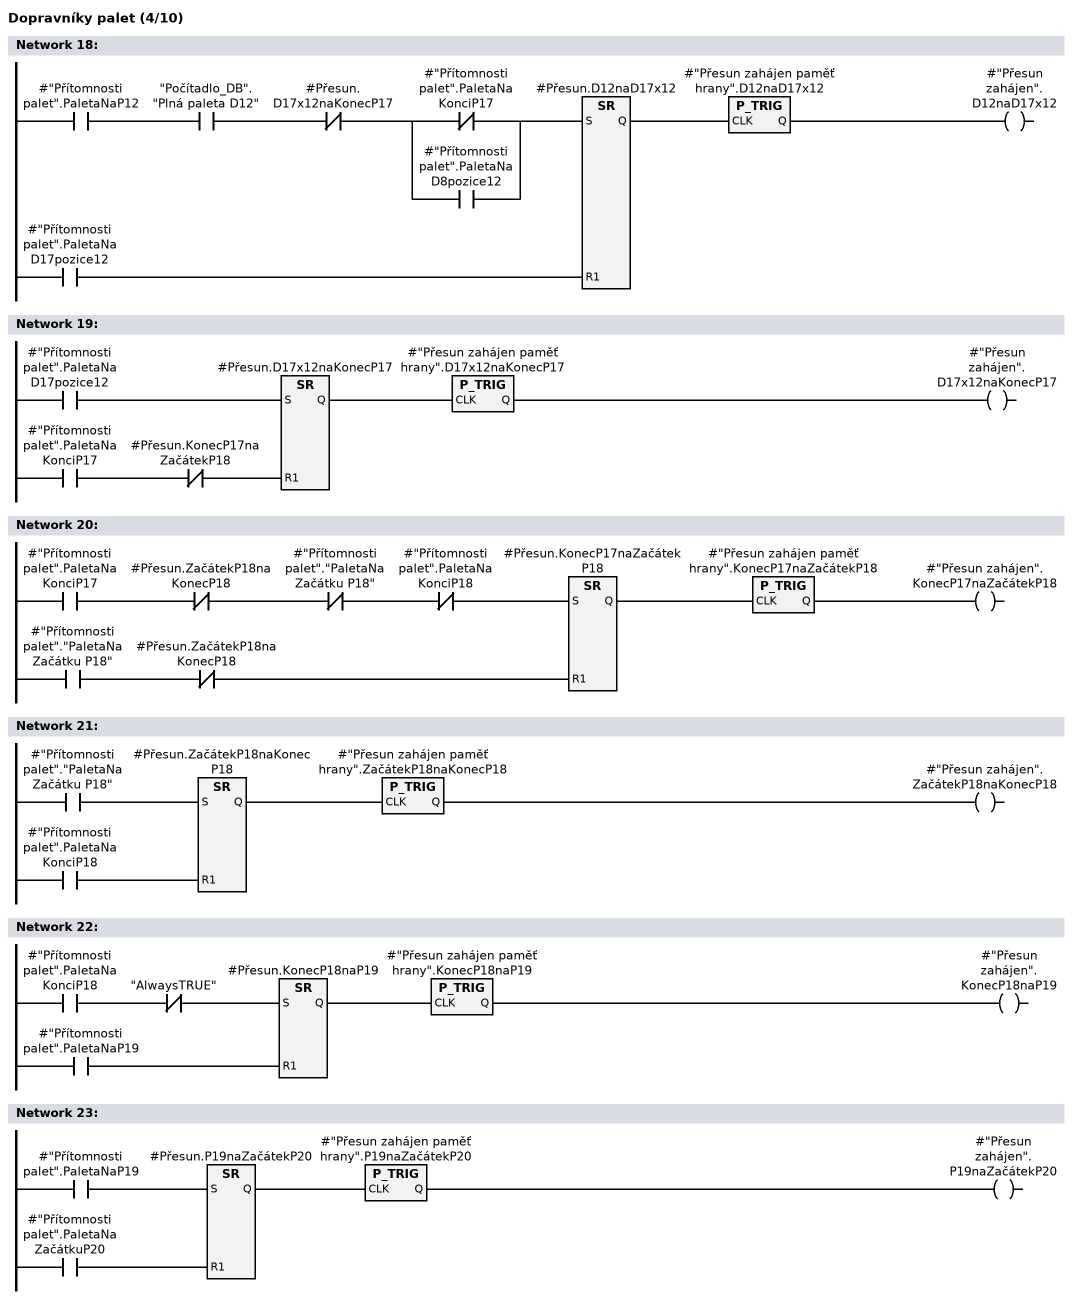
   RUNG wire#powerrail
      Contact( #"Přítomnosti palet".PaletaNaP12 )
      Contact( "Počítadlo_DB"."Plná paleta D12" )
      I_Contact( #Přesun.D17x12naKonecP17 )
      wire#w1
      I_Contact( #"Přítomnosti palet".PaletaNaKonciP17 )
      wire#w2
      S_SR(operand := #Přesun.D12naD17x12, r1 := wire#w3)
      P_Trig( #"Přesun zahájen paměť hrany".D12naD17x12 )
      Coil( #"Přesun zahájen".D12naD17x12 )
   END_RUNG
   RUNG wire#w1
      Contact( #"Přítomnosti palet".PaletaNaD8pozice12 )
   END_RUNG wire#w2
   RUNG wire#powerrail
      Contact( #"Přítomnosti palet".PaletaNaD17pozice12 )
   END_RUNG wire#w3
   // the same network as SCL:
   IF #"Přítomnosti palet".PaletaNaP12 AND "Počítadlo_DB"."Plná paleta D12" AND NOT #Přesun.D17x12naKonecP17 AND (NOT #"Přítomnosti palet".PaletaNaKonciP17 OR #"Přítomnosti palet".PaletaNaD8pozice12) THEN
       #Přesun.D12naD17x12 := TRUE;   // SR flip-flop
   END_IF;
   IF #"Přítomnosti palet".PaletaNaD17pozice12 THEN #Přesun.D12naD17x12 := FALSE; END_IF;
   #_w1 := #Přesun.D12naD17x12 AND NOT #"Přesun zahájen paměť hrany".D12naD17x12;   // rising edge
   #"Přesun zahájen paměť hrany".D12naD17x12 := #Přesun.D12naD17x12;
   #"Přesun zahájen".D12naD17x12 := #_w1;
END_REGION

REGION Network 19
   RUNG wire#powerrail
      Contact( #"Přítomnosti palet".PaletaNaD17pozice12 )
      S_SR(operand := #Přesun.D17x12naKonecP17, r1 := wire#w1)
      P_Trig( #"Přesun zahájen paměť hrany".D17x12naKonecP17 )
      Coil( #"Přesun zahájen".D17x12naKonecP17 )
   END_RUNG
   RUNG wire#powerrail
      Contact( #"Přítomnosti palet".PaletaNaKonciP17 )
      I_Contact( #Přesun.KonecP17naZačátekP18 )
   END_RUNG wire#w1
   // the same network as SCL:
   IF #"Přítomnosti palet".PaletaNaD17pozice12 THEN
       #Přesun.D17x12naKonecP17 := TRUE;   // SR flip-flop
   END_IF;
   IF #"Přítomnosti palet".PaletaNaKonciP17 AND NOT #Přesun.KonecP17naZačátekP18 THEN
       #Přesun.D17x12naKonecP17 := FALSE;
   END_IF;
   #_w1 := #Přesun.D17x12naKonecP17 AND NOT #"Přesun zahájen paměť hrany".D17x12naKonecP17;   // rising edge
   #"Přesun zahájen paměť hrany".D17x12naKonecP17 := #Přesun.D17x12naKonecP17;
   #"Přesun zahájen".D17x12naKonecP17 := #_w1;
END_REGION

REGION Network 20
   RUNG wire#powerrail
      Contact( #"Přítomnosti palet".PaletaNaKonciP17 )
      I_Contact( #Přesun.ZačátekP18naKonecP18 )
      I_Contact( #"Přítomnosti palet"."PaletaNaZačátku P18" )
      I_Contact( #"Přítomnosti palet".PaletaNaKonciP18 )
      S_SR(operand := #Přesun.KonecP17naZačátekP18, r1 := wire#w1)
      P_Trig( #"Přesun zahájen paměť hrany".KonecP17naZačátekP18 )
      Coil( #"Přesun zahájen".KonecP17naZačátekP18 )
   END_RUNG
   RUNG wire#powerrail
      Contact( #"Přítomnosti palet"."PaletaNaZačátku P18" )
      I_Contact( #Přesun.ZačátekP18naKonecP18 )
   END_RUNG wire#w1
   // the same network as SCL:
   IF #"Přítomnosti palet".PaletaNaKonciP17 AND NOT #Přesun.ZačátekP18naKonecP18 AND NOT #"Přítomnosti palet"."PaletaNaZačátku P18" AND NOT #"Přítomnosti palet".PaletaNaKonciP18 THEN
       #Přesun.KonecP17naZačátekP18 := TRUE;   // SR flip-flop
   END_IF;
   IF #"Přítomnosti palet"."PaletaNaZačátku P18" AND NOT #Přesun.ZačátekP18naKonecP18 THEN
       #Přesun.KonecP17naZačátekP18 := FALSE;
   END_IF;
   #_w1 := #Přesun.KonecP17naZačátekP18 AND NOT #"Přesun zahájen paměť hrany".KonecP17naZačátekP18;   // rising edge
   #"Přesun zahájen paměť hrany".KonecP17naZačátekP18 := #Přesun.KonecP17naZačátekP18;
   #"Přesun zahájen".KonecP17naZačátekP18 := #_w1;
END_REGION

REGION Network 21
   RUNG wire#powerrail
      Contact( #"Přítomnosti palet"."PaletaNaZačátku P18" )
      S_SR(operand := #Přesun.ZačátekP18naKonecP18, r1 := wire#w1)
      P_Trig( #"Přesun zahájen paměť hrany".ZačátekP18naKonecP18 )
      Coil( #"Přesun zahájen".ZačátekP18naKonecP18 )
   END_RUNG
   RUNG wire#powerrail
      Contact( #"Přítomnosti palet".PaletaNaKonciP18 )
   END_RUNG wire#w1
   // the same network as SCL:
   IF #"Přítomnosti palet"."PaletaNaZačátku P18" THEN
       #Přesun.ZačátekP18naKonecP18 := TRUE;   // SR flip-flop
   END_IF;
   IF #"Přítomnosti palet".PaletaNaKonciP18 THEN #Přesun.ZačátekP18naKonecP18 := FALSE; END_IF;
   #_w1 := #Přesun.ZačátekP18naKonecP18 AND NOT #"Přesun zahájen paměť hrany".ZačátekP18naKonecP18;   // rising edge
   #"Přesun zahájen paměť hrany".ZačátekP18naKonecP18 := #Přesun.ZačátekP18naKonecP18;
   #"Přesun zahájen".ZačátekP18naKonecP18 := #_w1;
END_REGION

REGION Network 22
   RUNG wire#powerrail
      Contact( #"Přítomnosti palet".PaletaNaKonciP18 )
      I_Contact( "AlwaysTRUE" )
      S_SR(operand := #Přesun.KonecP18naP19, r1 := wire#w1)
      P_Trig( #"Přesun zahájen paměť hrany".KonecP18naP19 )
      Coil( #"Přesun zahájen".KonecP18naP19 )
   END_RUNG
   RUNG wire#powerrail
      Contact( #"Přítomnosti palet".PaletaNaP19 )
   END_RUNG wire#w1
   // the same network as SCL:
   IF #"Přítomnosti palet".PaletaNaKonciP18 AND NOT "AlwaysTRUE" THEN
       #Přesun.KonecP18naP19 := TRUE;   // SR flip-flop
   END_IF;
   IF #"Přítomnosti palet".PaletaNaP19 THEN #Přesun.KonecP18naP19 := FALSE; END_IF;
   #_w1 := #Přesun.KonecP18naP19 AND NOT #"Přesun zahájen paměť hrany".KonecP18naP19;   // rising edge
   #"Přesun zahájen paměť hrany".KonecP18naP19 := #Přesun.KonecP18naP19;
   #"Přesun zahájen".KonecP18naP19 := #_w1;
END_REGION

REGION Network 23
   RUNG wire#powerrail
      Contact( #"Přítomnosti palet".PaletaNaP19 )
      S_SR(operand := #Přesun.P19naZačátekP20, r1 := wire#w1)
      P_Trig( #"Přesun zahájen paměť hrany".P19naZačátekP20 )
      Coil( #"Přesun zahájen".P19naZačátekP20 )
   END_RUNG
   RUNG wire#powerrail
      Contact( #"Přítomnosti palet".PaletaNaZačátkuP20 )
   END_RUNG wire#w1
   // the same network as SCL:
   IF #"Přítomnosti palet".PaletaNaP19 THEN
       #Přesun.P19naZačátekP20 := TRUE;   // SR flip-flop
   END_IF;
   IF #"Přítomnosti palet".PaletaNaZačátkuP20 THEN #Přesun.P19naZačátekP20 := FALSE; END_IF;
   #_w1 := #Přesun.P19naZačátekP20 AND NOT #"Přesun zahájen paměť hrany".P19naZačátekP20;   // rising edge
   #"Přesun zahájen paměť hrany".P19naZačátekP20 := #Přesun.P19naZačátekP20;
   #"Přesun zahájen".P19naZačátekP20 := #_w1;
END_REGION

REGION Network 24
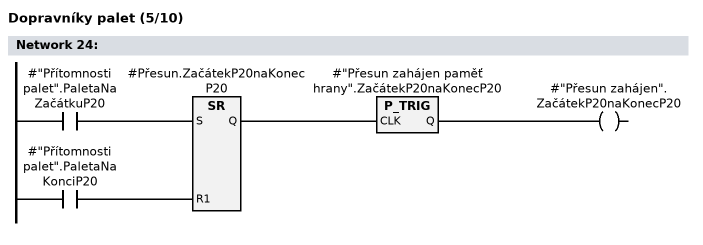
   RUNG wire#powerrail
      Contact( #"Přítomnosti palet".PaletaNaZačátkuP20 )
      S_SR(operand := #Přesun.ZačátekP20naKonecP20, r1 := wire#w1)
      P_Trig( #"Přesun zahájen paměť hrany".ZačátekP20naKonecP20 )
      Coil( #"Přesun zahájen".ZačátekP20naKonecP20 )
   END_RUNG
   RUNG wire#powerrail
      Contact( #"Přítomnosti palet".PaletaNaKonciP20 )
   END_RUNG wire#w1
   // the same network as SCL:
   IF #"Přítomnosti palet".PaletaNaZačátkuP20 THEN
       #Přesun.ZačátekP20naKonecP20 := TRUE;   // SR flip-flop
   END_IF;
   IF #"Přítomnosti palet".PaletaNaKonciP20 THEN #Přesun.ZačátekP20naKonecP20 := FALSE; END_IF;
   #_w1 := #Přesun.ZačátekP20naKonecP20 AND NOT #"Přesun zahájen paměť hrany".ZačátekP20naKonecP20;   // rising edge
   #"Přesun zahájen paměť hrany".ZačátekP20naKonecP20 := #Přesun.ZačátekP20naKonecP20;
   #"Přesun zahájen".ZačátekP20naKonecP20 := #_w1;
END_REGION

REGION Network 25
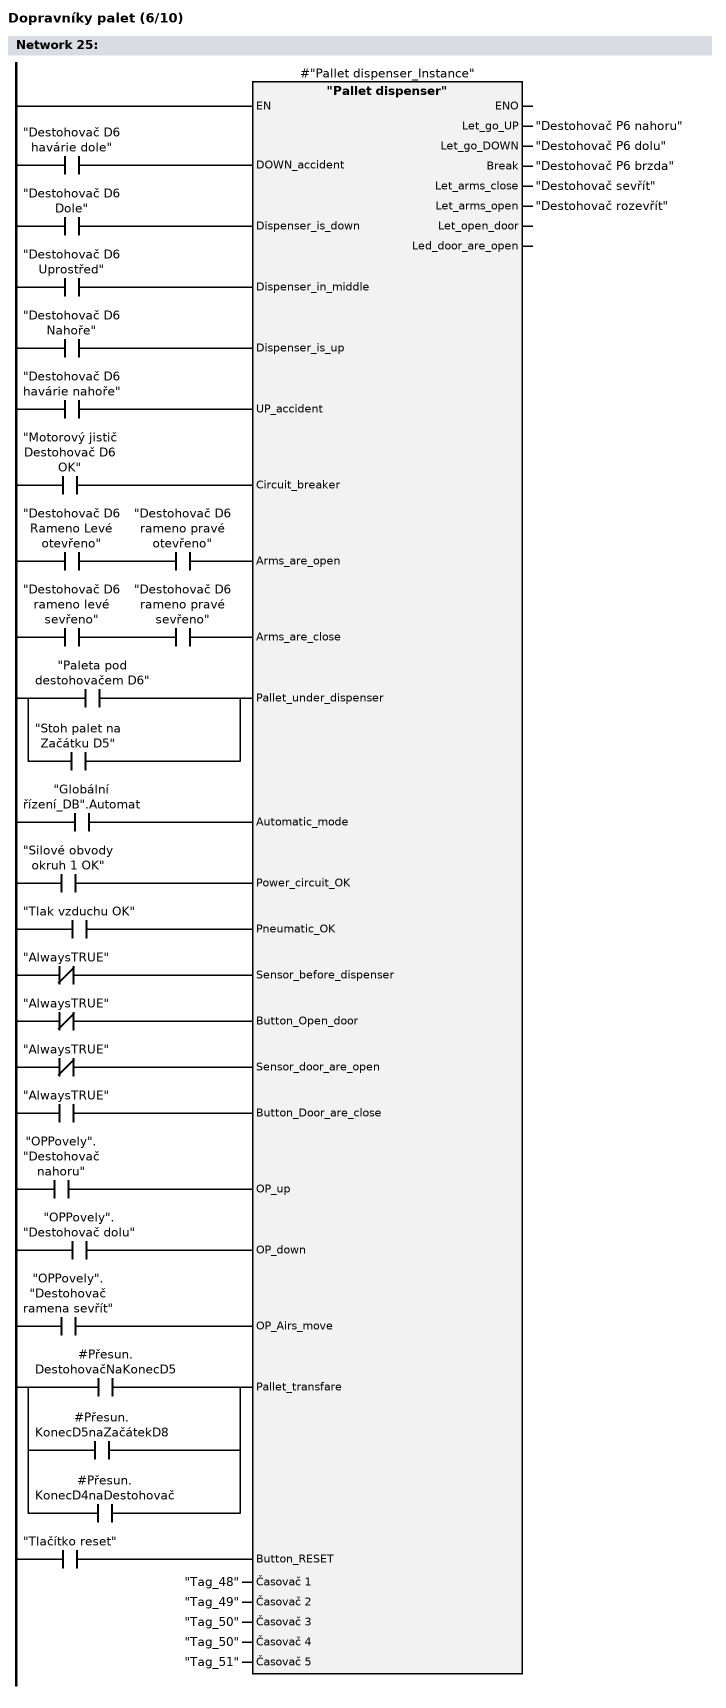
   RUNG wire#powerrail
      #"Pallet dispenser_Instance"(DOWN_accident := wire#w1, Dispenser_is_down := wire#w2, Dispenser_in_middle := wire#w3, Dispenser_is_up := wire#w4, UP_accident := wire#w5, Circuit_breaker := wire#w6, Arms_are_open := wire#w7, Arms_are_close := wire#w8, Pallet_under_dispenser := wire#w9, Automatic_mode := wire#w10, Power_circuit_OK := wire#w11, Pneumatic_OK := wire#w12, Sensor_before_dispenser := wire#w13, Button_Open_door := wire#w14, Sensor_door_are_open := wire#w15, Button_Door_are_close := wire#w16, OP_up := wire#w17, OP_down := wire#w18, OP_Airs_move := wire#w19, Pallet_transfare := wire#w20, Button_RESET := wire#w21, "Časovač 1" := "Tag_48", "Časovač 2" := "Tag_49", "Časovač 3" := "Tag_50", "Časovač 4" := "Tag_50", "Časovač 5" := "Tag_51", Let_go_UP => "Destohovač P6 nahoru", Let_go_DOWN => "Destohovač P6 dolu", Break => "Destohovač P6 brzda", Let_arms_close => "Destohovač sevřít", Let_arms_open => "Destohovač rozevřít", Let_open_door =>, Led_door_are_open =>)
   END_RUNG
   RUNG wire#powerrail
      Contact( "Destohovač D6 havárie dole" )
   END_RUNG wire#w1
   RUNG wire#powerrail
      Contact( "Destohovač D6 Dole" )
   END_RUNG wire#w2
   RUNG wire#powerrail
      Contact( "Destohovač D6 Uprostřed" )
   END_RUNG wire#w3
   RUNG wire#powerrail
      Contact( "Destohovač D6 Nahoře" )
   END_RUNG wire#w4
   RUNG wire#powerrail
      Contact( "Destohovač D6 havárie nahoře" )
   END_RUNG wire#w5
   RUNG wire#powerrail
      Contact( "Motorový jistič Destohovač D6 OK" )
   END_RUNG wire#w6
   RUNG wire#powerrail
      Contact( "Destohovač D6 Rameno Levé otevřeno" )
      Contact( "Destohovač D6 rameno pravé otevřeno" )
   END_RUNG wire#w7
   RUNG wire#powerrail
      Contact( "Destohovač D6 rameno levé sevřeno" )
      Contact( "Destohovač D6 rameno pravé sevřeno" )
   END_RUNG wire#w8
   RUNG wire#powerrail
      Contact( "Paleta pod destohovačem D6" )
   END_RUNG wire#w9
   RUNG wire#powerrail
      Contact( "Stoh palet na Začátku D5" )
   END_RUNG wire#w9
   RUNG wire#powerrail
      Contact( "Globální řízení_DB".Automat )
   END_RUNG wire#w10
   RUNG wire#powerrail
      Contact( "Silové obvody okruh 1 OK" )
   END_RUNG wire#w11
   RUNG wire#powerrail
      Contact( "Tlak vzduchu OK" )
   END_RUNG wire#w12
   RUNG wire#powerrail
      I_Contact( "AlwaysTRUE" )
   END_RUNG wire#w13
   RUNG wire#powerrail
      I_Contact( "AlwaysTRUE" )
   END_RUNG wire#w14
   RUNG wire#powerrail
      I_Contact( "AlwaysTRUE" )
   END_RUNG wire#w15
   RUNG wire#powerrail
      Contact( "AlwaysTRUE" )
   END_RUNG wire#w16
   RUNG wire#powerrail
      Contact( "OPPovely"."Destohovač nahoru" )
   END_RUNG wire#w17
   RUNG wire#powerrail
      Contact( "OPPovely"."Destohovač dolu" )
   END_RUNG wire#w18
   RUNG wire#powerrail
      Contact( "OPPovely"."Destohovač ramena sevřít" )
   END_RUNG wire#w19
   RUNG wire#powerrail
      Contact( #Přesun.DestohovačNaKonecD5 )
   END_RUNG wire#w20
   RUNG wire#powerrail
      Contact( #Přesun.KonecD5naZačátekD8 )
   END_RUNG wire#w20
   RUNG wire#powerrail
      Contact( #Přesun.KonecD4naDestohovač )
   END_RUNG wire#w20
   RUNG wire#powerrail
      Contact( "Tlačítko reset" )
   END_RUNG wire#w21
   // the same network as SCL:
   #"Pallet dispenser_Instance"(DOWN_accident := "Destohovač D6 havárie dole",   // "Pallet dispenser"
                           Dispenser_is_down := "Destohovač D6 Dole",
                           Dispenser_in_middle := "Destohovač D6 Uprostřed",
                           Dispenser_is_up := "Destohovač D6 Nahoře",
                           UP_accident := "Destohovač D6 havárie nahoře",
                           Circuit_breaker := "Motorový jistič Destohovač D6 OK",
                           Arms_are_open := "Destohovač D6 Rameno Levé otevřeno" AND "Destohovač D6 rameno pravé otevřeno",
                           Arms_are_close := "Destohovač D6 rameno levé sevřeno" AND "Destohovač D6 rameno pravé sevřeno",
                           Pallet_under_dispenser := "Paleta pod destohovačem D6" OR "Stoh palet na Začátku D5",
                           Automatic_mode := "Globální řízení_DB".Automat,
                           Power_circuit_OK := "Silové obvody okruh 1 OK",
                           Pneumatic_OK := "Tlak vzduchu OK",
                           Sensor_before_dispenser := NOT "AlwaysTRUE",
                           Button_Open_door := NOT "AlwaysTRUE",
                           Sensor_door_are_open := NOT "AlwaysTRUE",
                           Button_Door_are_close := "AlwaysTRUE",
                           OP_up := "OPPovely"."Destohovač nahoru",
                           OP_down := "OPPovely"."Destohovač dolu",
                           OP_Airs_move := "OPPovely"."Destohovač ramena sevřít",
                           Pallet_transfare := #Přesun.DestohovačNaKonecD5 OR #Přesun.KonecD5naZačátekD8 OR #Přesun.KonecD4naDestohovač,
                           Button_RESET := "Tlačítko reset",
                           "Časovač 1" := "Tag_48",
                           "Časovač 2" := "Tag_49",
                           "Časovač 3" := "Tag_50",
                           "Časovač 4" := "Tag_50",
                           "Časovač 5" := "Tag_51",
                           Let_go_UP => "Destohovač P6 nahoru",
                           Let_go_DOWN => "Destohovač P6 dolu",
                           Break => "Destohovač P6 brzda",
                           Let_arms_close => "Destohovač sevřít",
                           Let_arms_open => "Destohovač rozevřít");
END_REGION

REGION Network 26
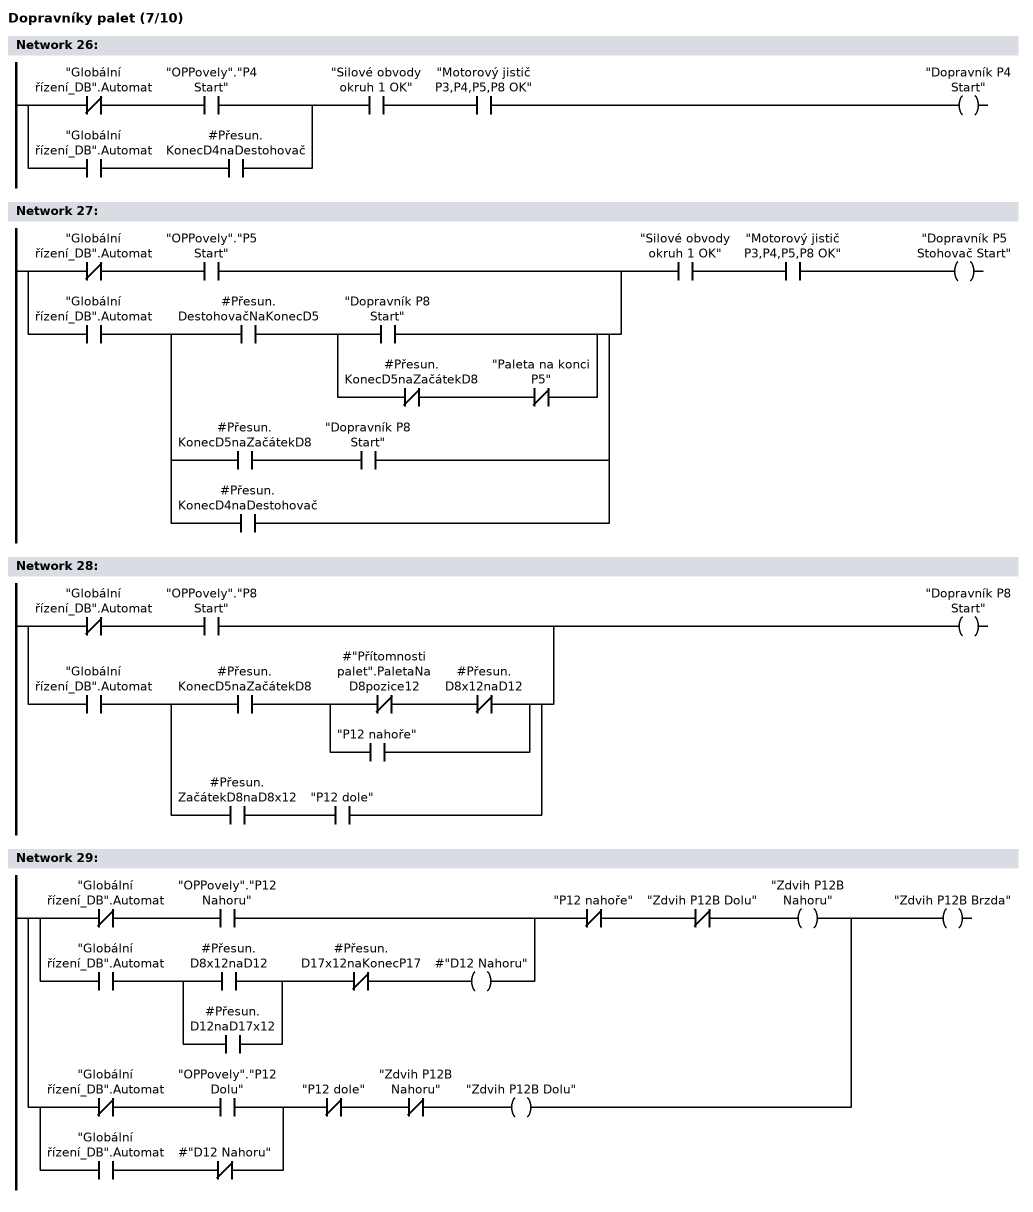
   RUNG wire#powerrail
      I_Contact( "Globální řízení_DB".Automat )
      Contact( "OPPovely"."P4 Start" )
      wire#w1
      Contact( "Silové obvody okruh 1 OK" )
      Contact( "Motorový jistič P3,P4,P5,P8 OK" )
      Coil( "Dopravník P4 Start" )
   END_RUNG
   RUNG wire#powerrail
      Contact( "Globální řízení_DB".Automat )
      Contact( #Přesun.KonecD4naDestohovač )
   END_RUNG wire#w1
   // the same network as SCL:
   "Dopravník P4 Start" := ((NOT "Globální řízení_DB".Automat AND "OPPovely"."P4 Start") OR ("Globální řízení_DB".Automat AND #Přesun.KonecD4naDestohovač)) AND "Silové obvody okruh 1 OK" AND "Motorový jistič P3,P4,P5,P8 OK";
END_REGION

REGION Network 27
   RUNG wire#powerrail
      I_Contact( "Globální řízení_DB".Automat )
      Contact( "OPPovely"."P5 Start" )
      wire#w1
      Contact( "Silové obvody okruh 1 OK" )
      Contact( "Motorový jistič P3,P4,P5,P8 OK" )
      Coil( "Dopravník P5 Stohovač Start" )
   END_RUNG
   RUNG wire#powerrail
      Contact( "Globální řízení_DB".Automat )
      wire#w2
      Contact( #Přesun.DestohovačNaKonecD5 )
      wire#w3
      Contact( "Dopravník P8 Start" )
   END_RUNG wire#w1
   RUNG wire#w3
      I_Contact( #Přesun.KonecD5naZačátekD8 )
      I_Contact( "Paleta na konci P5" )
   END_RUNG wire#w1
   RUNG wire#w2
      Contact( #Přesun.KonecD5naZačátekD8 )
      Contact( "Dopravník P8 Start" )
   END_RUNG wire#w1
   RUNG wire#w2
      Contact( #Přesun.KonecD4naDestohovač )
   END_RUNG wire#w1
   // the same network as SCL:
   "Dopravník P5 Stohovač Start" := ((NOT "Globální řízení_DB".Automat AND "OPPovely"."P5 Start") OR ("Globální řízení_DB".Automat AND ((#Přesun.DestohovačNaKonecD5 AND ("Dopravník P8 Start" OR (NOT #Přesun.KonecD5naZačátekD8 AND NOT "Paleta na konci P5"))) OR (#Přesun.KonecD5naZačátekD8 AND "Dopravník P8 Start") OR #Přesun.KonecD4naDestohovač))) AND "Silové obvody okruh 1 OK" AND "Motorový jistič P3,P4,P5,P8 OK";
END_REGION

REGION Network 28
   RUNG wire#powerrail
      I_Contact( "Globální řízení_DB".Automat )
      Contact( "OPPovely"."P8 Start" )
      wire#w1
      Coil( "Dopravník P8 Start" )
   END_RUNG
   RUNG wire#powerrail
      Contact( "Globální řízení_DB".Automat )
      wire#w2
      Contact( #Přesun.KonecD5naZačátekD8 )
      wire#w3
      I_Contact( #"Přítomnosti palet".PaletaNaD8pozice12 )
      I_Contact( #Přesun.D8x12naD12 )
   END_RUNG wire#w1
   RUNG wire#w3
      Contact( "P12 nahoře" )
   END_RUNG wire#w1
   RUNG wire#w2
      Contact( #Přesun.ZačátekD8naD8x12 )
      Contact( "P12 dole" )
   END_RUNG wire#w1
   // the same network as SCL:
   "Dopravník P8 Start" := (NOT "Globální řízení_DB".Automat AND "OPPovely"."P8 Start") OR ("Globální řízení_DB".Automat AND ((#Přesun.KonecD5naZačátekD8 AND ((NOT #"Přítomnosti palet".PaletaNaD8pozice12 AND NOT #Přesun.D8x12naD12) OR "P12 nahoře")) OR (#Přesun.ZačátekD8naD8x12 AND "P12 dole")));
END_REGION

REGION Network 29
   RUNG wire#powerrail
      I_Contact( "Globální řízení_DB".Automat )
      Contact( "OPPovely"."P12 Nahoru" )
      wire#w1
      I_Contact( "P12 nahoře" )
      I_Contact( "Zdvih P12B Dolu" )
      Coil( "Zdvih P12B Nahoru" )
      wire#w4
      Coil( "Zdvih P12B Brzda" )
   END_RUNG
   RUNG wire#powerrail
      Contact( "Globální řízení_DB".Automat )
      wire#w2
      Contact( #Přesun.D8x12naD12 )
      wire#w3
      I_Contact( #Přesun.D17x12naKonecP17 )
      Coil( #"D12 Nahoru" )
   END_RUNG wire#w1
   RUNG wire#w2
      Contact( #Přesun.D12naD17x12 )
   END_RUNG wire#w3
   RUNG wire#powerrail
      I_Contact( "Globální řízení_DB".Automat )
      Contact( "OPPovely"."P12 Dolu" )
      wire#w5
      I_Contact( "P12 dole" )
      I_Contact( "Zdvih P12B Nahoru" )
      Coil( "Zdvih P12B Dolu" )
   END_RUNG wire#w4
   RUNG wire#powerrail
      Contact( "Globální řízení_DB".Automat )
      I_Contact( #"D12 Nahoru" )
   END_RUNG wire#w5
   // the same network as SCL:
   #"D12 Nahoru" := "Globální řízení_DB".Automat AND (#Přesun.D8x12naD12 OR #Přesun.D12naD17x12) AND NOT #Přesun.D17x12naKonecP17;
   "Zdvih P12B Nahoru" := ((NOT "Globální řízení_DB".Automat AND "OPPovely"."P12 Nahoru") OR #"D12 Nahoru") AND NOT "P12 nahoře" AND NOT "Zdvih P12B Dolu";
   "Zdvih P12B Dolu" := ((NOT "Globální řízení_DB".Automat AND "OPPovely"."P12 Dolu") OR ("Globální řízení_DB".Automat AND NOT #"D12 Nahoru")) AND NOT "P12 dole" AND NOT "Zdvih P12B Nahoru";
   "Zdvih P12B Brzda" := "Zdvih P12B Nahoru" OR "Zdvih P12B Dolu";
END_REGION

REGION Network 30
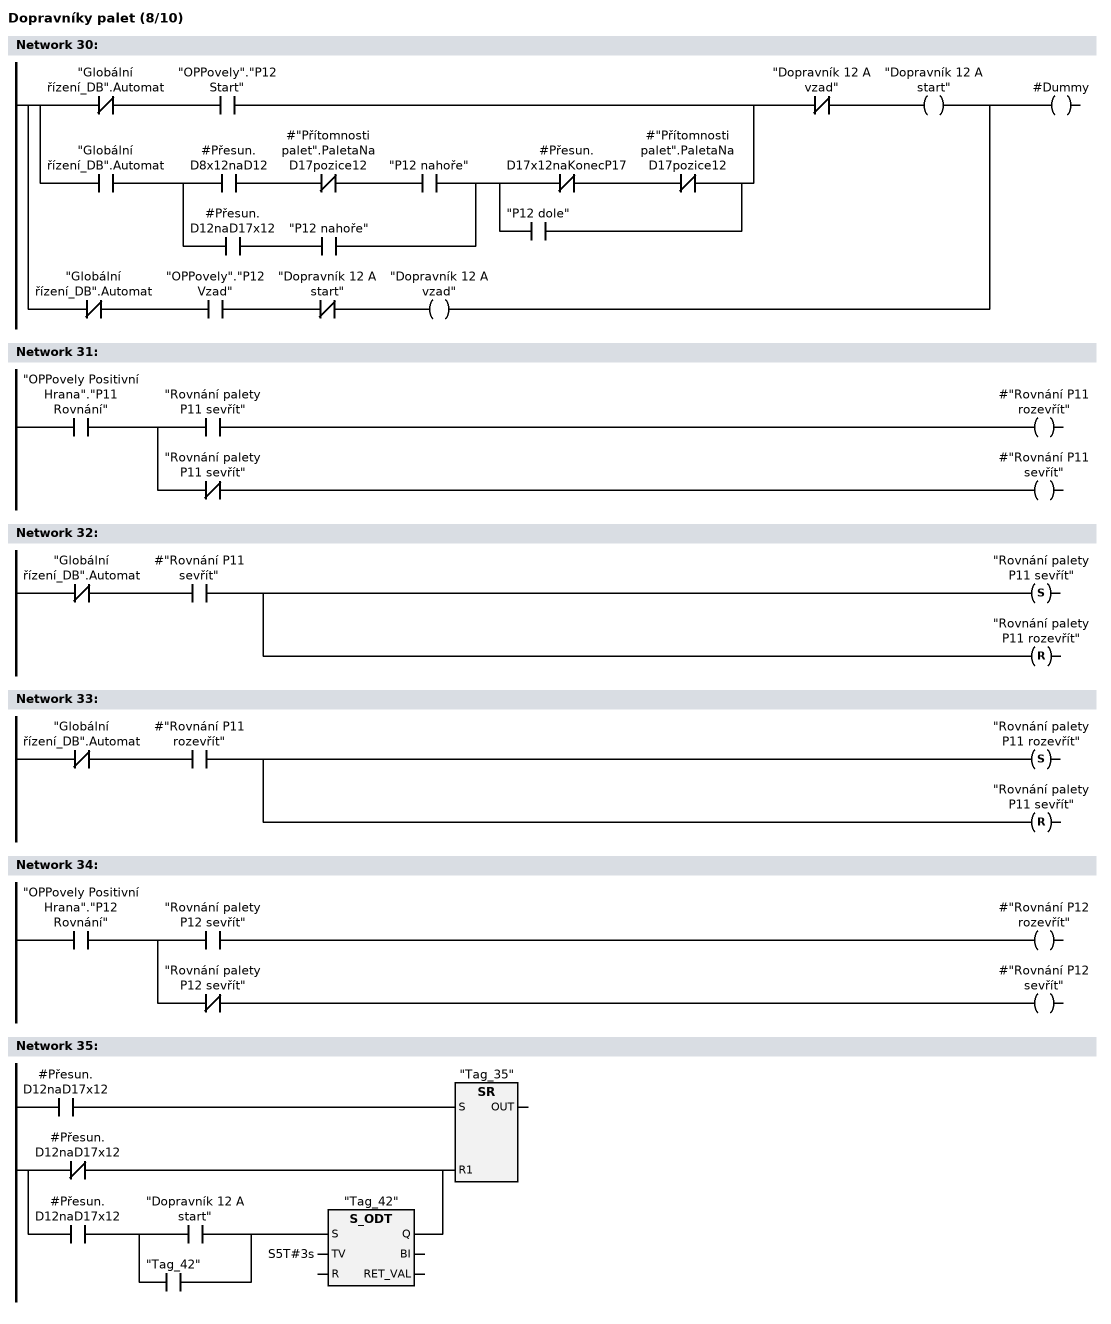
   RUNG wire#powerrail
      I_Contact( "Globální řízení_DB".Automat )
      Contact( "OPPovely"."P12 Start" )
      wire#w1
      I_Contact( "Dopravník 12 A vzad" )
      Coil( "Dopravník 12 A start" )
      wire#w4
      Coil( #Dummy )
   END_RUNG
   RUNG wire#powerrail
      Contact( "Globální řízení_DB".Automat )
      wire#w2
      Contact( #Přesun.D8x12naD12 )
      I_Contact( #"Přítomnosti palet".PaletaNaD17pozice12 )
      Contact( "P12 nahoře" )
      wire#w3
      I_Contact( #Přesun.D17x12naKonecP17 )
      I_Contact( #"Přítomnosti palet".PaletaNaD17pozice12 )
   END_RUNG wire#w1
   RUNG wire#w2
      Contact( #Přesun.D12naD17x12 )
      Contact( "P12 nahoře" )
   END_RUNG wire#w3
   RUNG wire#w3
      Contact( "P12 dole" )
   END_RUNG wire#w1
   RUNG wire#powerrail
      I_Contact( "Globální řízení_DB".Automat )
      Contact( "OPPovely"."P12 Vzad" )
      I_Contact( "Dopravník 12 A start" )
      Coil( "Dopravník 12 A vzad" )
   END_RUNG wire#w4
   // the same network as SCL:
   "Dopravník 12 A start" := ((NOT "Globální řízení_DB".Automat AND "OPPovely"."P12 Start") OR ("Globální řízení_DB".Automat AND ((#Přesun.D8x12naD12 AND NOT #"Přítomnosti palet".PaletaNaD17pozice12 AND "P12 nahoře") OR (#Přesun.D12naD17x12 AND "P12 nahoře")) AND ((NOT #Přesun.D17x12naKonecP17 AND NOT #"Přítomnosti palet".PaletaNaD17pozice12) OR "P12 dole"))) AND NOT "Dopravník 12 A vzad";
   "Dopravník 12 A vzad" := NOT "Globální řízení_DB".Automat AND "OPPovely"."P12 Vzad" AND NOT "Dopravník 12 A start";
   #Dummy := "Dopravník 12 A start" OR "Dopravník 12 A vzad";
END_REGION

REGION Network 31
   RUNG wire#powerrail
      Contact( "OPPovely Positivní Hrana"."P11 Rovnání" )
      wire#w1
      Contact( "Rovnání palety P11 sevřít" )
      Coil( #"Rovnání P11 rozevřít" )
   END_RUNG
   RUNG wire#w1
      I_Contact( "Rovnání palety P11 sevřít" )
      Coil( #"Rovnání P11 sevřít" )
   END_RUNG
   // the same network as SCL:
   #"Rovnání P11 rozevřít" := "OPPovely Positivní Hrana"."P11 Rovnání" AND "Rovnání palety P11 sevřít";
   #"Rovnání P11 sevřít" := "OPPovely Positivní Hrana"."P11 Rovnání" AND NOT "Rovnání palety P11 sevřít";
END_REGION

REGION Network 32
   RUNG wire#powerrail
      I_Contact( "Globální řízení_DB".Automat )
      Contact( #"Rovnání P11 sevřít" )
      wire#w1
      S_Coil( "Rovnání palety P11 sevřít" )
   END_RUNG
   RUNG wire#w1
      R_Coil( "Rovnání palety P11 rozevřít" )
   END_RUNG
   // the same network as SCL:
   IF NOT "Globální řízení_DB".Automat AND #"Rovnání P11 sevřít" THEN
       "Rovnání palety P11 sevřít" := TRUE;
       "Rovnání palety P11 rozevřít" := FALSE;
   END_IF;
END_REGION

REGION Network 33
   RUNG wire#powerrail
      I_Contact( "Globální řízení_DB".Automat )
      Contact( #"Rovnání P11 rozevřít" )
      wire#w1
      S_Coil( "Rovnání palety P11 rozevřít" )
   END_RUNG
   RUNG wire#w1
      R_Coil( "Rovnání palety P11 sevřít" )
   END_RUNG
   // the same network as SCL:
   IF NOT "Globální řízení_DB".Automat AND #"Rovnání P11 rozevřít" THEN
       "Rovnání palety P11 rozevřít" := TRUE;
       "Rovnání palety P11 sevřít" := FALSE;
   END_IF;
END_REGION

REGION Network 34
   RUNG wire#powerrail
      Contact( "OPPovely Positivní Hrana"."P12 Rovnání" )
      wire#w1
      Contact( "Rovnání palety P12 sevřít" )
      Coil( #"Rovnání P12 rozevřít" )
   END_RUNG
   RUNG wire#w1
      I_Contact( "Rovnání palety P12 sevřít" )
      Coil( #"Rovnání P12 sevřít" )
   END_RUNG
   // the same network as SCL:
   #"Rovnání P12 rozevřít" := "OPPovely Positivní Hrana"."P12 Rovnání" AND "Rovnání palety P12 sevřít";
   #"Rovnání P12 sevřít" := "OPPovely Positivní Hrana"."P12 Rovnání" AND NOT "Rovnání palety P12 sevřít";
END_REGION

REGION Network 35
   RUNG wire#powerrail
      Contact( #Přesun.D12naD17x12 )
      S_SR(operand := "Tag_35", r1 := wire#w3)
   END_RUNG
   RUNG wire#powerrail
      I_Contact( #Přesun.D12naD17x12 )
   END_RUNG wire#w3
   RUNG wire#powerrail
      Contact( #Přesun.D12naD17x12 )
      wire#w1
      Contact( "Dopravník 12 A start" )
      wire#w2
      S_ODT(T_NO := "Tag_42", TV := S5T#3s, R :=, BI =>, RET_VAL =>)
   END_RUNG wire#w3
   RUNG wire#w1
      Contact( "Tag_42" )
   END_RUNG wire#w2
   // the same network as SCL:
   #_w2 := #Přesun.D12naD17x12;
   #_w3 := NOT #Přesun.D12naD17x12;
   #_s5time1 := S_ODT(T_NO := "Tag_42",
                      S := #Přesun.D12naD17x12 AND ("Dopravník 12 A start" OR "Tag_42"),
                      TV := S5T#3s,
                      Q => #_w1);
   IF #_w2 THEN
       "Tag_35" := TRUE;   // SR flip-flop
   END_IF;
   IF #_w3 OR #_w1 THEN "Tag_35" := FALSE; END_IF;
END_REGION

REGION Network 36
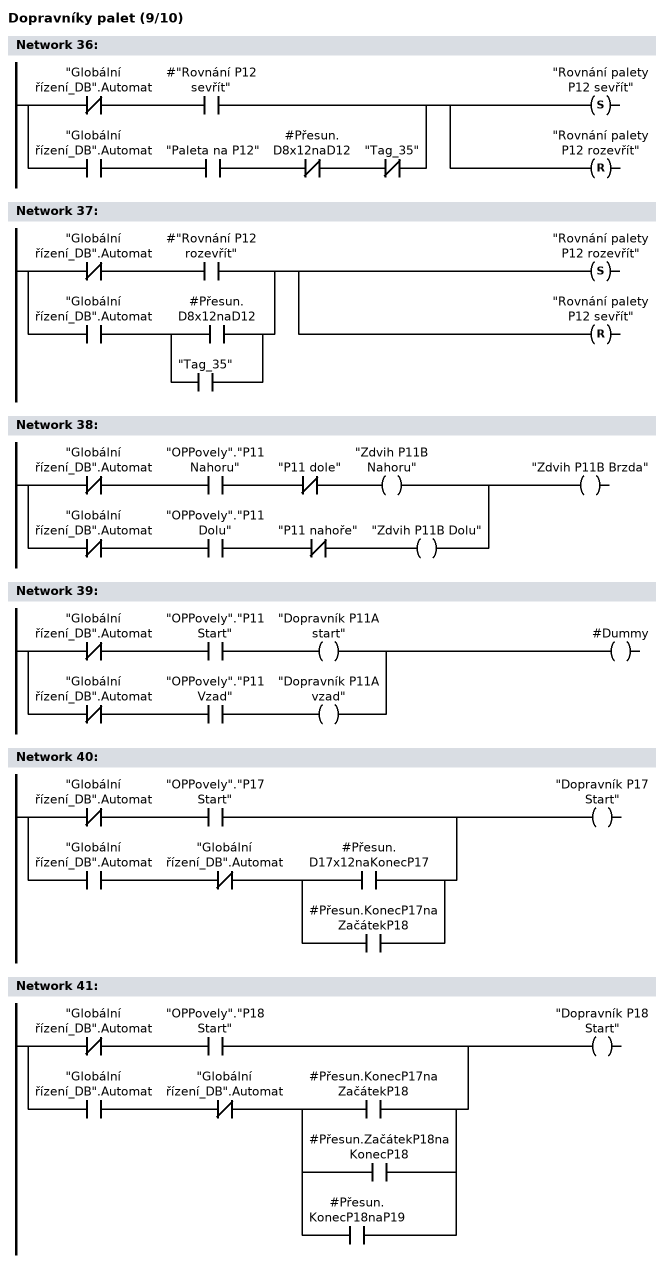
   RUNG wire#powerrail
      I_Contact( "Globální řízení_DB".Automat )
      Contact( #"Rovnání P12 sevřít" )
      wire#w1
      S_Coil( "Rovnání palety P12 sevřít" )
   END_RUNG
   RUNG wire#powerrail
      Contact( "Globální řízení_DB".Automat )
      Contact( "Paleta na P12" )
      I_Contact( #Přesun.D8x12naD12 )
      I_Contact( "Tag_35" )
   END_RUNG wire#w1
   RUNG wire#w1
      R_Coil( "Rovnání palety P12 rozevřít" )
   END_RUNG
   // the same network as SCL:
   IF (NOT "Globální řízení_DB".Automat AND #"Rovnání P12 sevřít") OR ("Globální řízení_DB".Automat AND "Paleta na P12" AND NOT #Přesun.D8x12naD12 AND NOT "Tag_35") THEN
       "Rovnání palety P12 sevřít" := TRUE;
       "Rovnání palety P12 rozevřít" := FALSE;
   END_IF;
END_REGION

REGION Network 37
   RUNG wire#powerrail
      I_Contact( "Globální řízení_DB".Automat )
      Contact( #"Rovnání P12 rozevřít" )
      wire#w1
      S_Coil( "Rovnání palety P12 rozevřít" )
   END_RUNG
   RUNG wire#powerrail
      Contact( "Globální řízení_DB".Automat )
      wire#w2
      Contact( #Přesun.D8x12naD12 )
   END_RUNG wire#w1
   RUNG wire#w2
      Contact( "Tag_35" )
   END_RUNG wire#w1
   RUNG wire#w1
      R_Coil( "Rovnání palety P12 sevřít" )
   END_RUNG
   // the same network as SCL:
   IF (NOT "Globální řízení_DB".Automat AND #"Rovnání P12 rozevřít") OR ("Globální řízení_DB".Automat AND (#Přesun.D8x12naD12 OR "Tag_35")) THEN
       "Rovnání palety P12 rozevřít" := TRUE;
       "Rovnání palety P12 sevřít" := FALSE;
   END_IF;
END_REGION

REGION Network 38
   RUNG wire#powerrail
      I_Contact( "Globální řízení_DB".Automat )
      Contact( "OPPovely"."P11 Nahoru" )
      I_Contact( "P11 dole" )
      Coil( "Zdvih P11B Nahoru" )
      wire#w1
      Coil( "Zdvih P11B Brzda" )
   END_RUNG
   RUNG wire#powerrail
      I_Contact( "Globální řízení_DB".Automat )
      Contact( "OPPovely"."P11 Dolu" )
      I_Contact( "P11 nahoře" )
      Coil( "Zdvih P11B Dolu" )
   END_RUNG wire#w1
   // the same network as SCL:
   "Zdvih P11B Nahoru" := NOT "Globální řízení_DB".Automat AND "OPPovely"."P11 Nahoru" AND NOT "P11 dole";
   "Zdvih P11B Dolu" := NOT "Globální řízení_DB".Automat AND "OPPovely"."P11 Dolu" AND NOT "P11 nahoře";
   "Zdvih P11B Brzda" := "Zdvih P11B Nahoru" OR "Zdvih P11B Dolu";
END_REGION

REGION Network 39
   RUNG wire#powerrail
      I_Contact( "Globální řízení_DB".Automat )
      Contact( "OPPovely"."P11 Start" )
      Coil( "Dopravník P11A start" )
      wire#w1
      Coil( #Dummy )
   END_RUNG
   RUNG wire#powerrail
      I_Contact( "Globální řízení_DB".Automat )
      Contact( "OPPovely"."P11 Vzad" )
      Coil( "Dopravník P11A vzad" )
   END_RUNG wire#w1
   // the same network as SCL:
   "Dopravník P11A start" := NOT "Globální řízení_DB".Automat AND "OPPovely"."P11 Start";
   "Dopravník P11A vzad" := NOT "Globální řízení_DB".Automat AND "OPPovely"."P11 Vzad";
   #Dummy := "Dopravník P11A start" OR "Dopravník P11A vzad";
END_REGION

REGION Network 40
   RUNG wire#powerrail
      I_Contact( "Globální řízení_DB".Automat )
      Contact( "OPPovely"."P17 Start" )
      wire#w1
      Coil( "Dopravník P17 Start" )
   END_RUNG
   RUNG wire#powerrail
      Contact( "Globální řízení_DB".Automat )
      I_Contact( "Globální řízení_DB".Automat )
      wire#w2
      Contact( #Přesun.D17x12naKonecP17 )
   END_RUNG wire#w1
   RUNG wire#w2
      Contact( #Přesun.KonecP17naZačátekP18 )
   END_RUNG wire#w1
   // the same network as SCL:
   "Dopravník P17 Start" := (NOT "Globální řízení_DB".Automat AND "OPPovely"."P17 Start") OR ("Globální řízení_DB".Automat AND NOT "Globální řízení_DB".Automat AND (#Přesun.D17x12naKonecP17 OR #Přesun.KonecP17naZačátekP18));
END_REGION

REGION Network 41
   RUNG wire#powerrail
      I_Contact( "Globální řízení_DB".Automat )
      Contact( "OPPovely"."P18 Start" )
      wire#w1
      Coil( "Dopravník P18 Start" )
   END_RUNG
   RUNG wire#powerrail
      Contact( "Globální řízení_DB".Automat )
      I_Contact( "Globální řízení_DB".Automat )
      wire#w2
      Contact( #Přesun.KonecP17naZačátekP18 )
   END_RUNG wire#w1
   RUNG wire#w2
      Contact( #Přesun.ZačátekP18naKonecP18 )
   END_RUNG wire#w1
   RUNG wire#w2
      Contact( #Přesun.KonecP18naP19 )
   END_RUNG wire#w1
   // the same network as SCL:
   "Dopravník P18 Start" := (NOT "Globální řízení_DB".Automat AND "OPPovely"."P18 Start") OR ("Globální řízení_DB".Automat AND NOT "Globální řízení_DB".Automat AND (#Přesun.KonecP17naZačátekP18 OR #Přesun.ZačátekP18naKonecP18 OR #Přesun.KonecP18naP19));
END_REGION

REGION Network 42
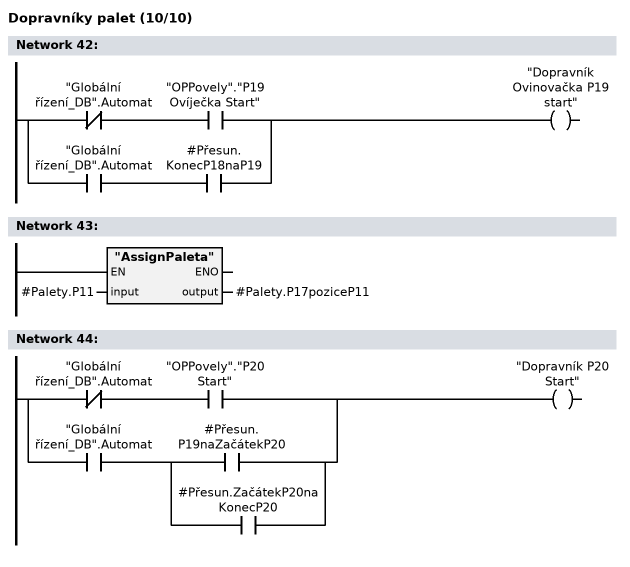
   RUNG wire#powerrail
      I_Contact( "Globální řízení_DB".Automat )
      Contact( "OPPovely"."P19 Ovíječka Start" )
      wire#w1
      Coil( "Dopravník Ovinovačka P19 start" )
   END_RUNG
   RUNG wire#powerrail
      Contact( "Globální řízení_DB".Automat )
      Contact( #Přesun.KonecP18naP19 )
   END_RUNG wire#w1
   // the same network as SCL:
   "Dopravník Ovinovačka P19 start" := (NOT "Globální řízení_DB".Automat AND "OPPovely"."P19 Ovíječka Start") OR ("Globální řízení_DB".Automat AND #Přesun.KonecP18naP19);
END_REGION

REGION Network 43
   RUNG wire#powerrail
      "AssignPaleta"(input := #Palety.P11, output => #Palety.P17poziceP11)
   END_RUNG
   // the same network as SCL:
   "AssignPaleta"(input := #Palety.P11, output => #Palety.P17poziceP11);
END_REGION

REGION Network 44
   RUNG wire#powerrail
      I_Contact( "Globální řízení_DB".Automat )
      Contact( "OPPovely"."P20 Start" )
      wire#w1
      Coil( "Dopravník P20 Start" )
   END_RUNG
   RUNG wire#powerrail
      Contact( "Globální řízení_DB".Automat )
      wire#w2
      Contact( #Přesun.P19naZačátekP20 )
   END_RUNG wire#w1
   RUNG wire#w2
      Contact( #Přesun.ZačátekP20naKonecP20 )
   END_RUNG wire#w1
   // the same network as SCL:
   "Dopravník P20 Start" := (NOT "Globální řízení_DB".Automat AND "OPPovely"."P20 Start") OR ("Globální řízení_DB".Automat AND (#Přesun.P19naZačátekP20 OR #Přesun.ZačátekP20naKonecP20));
END_REGION
END_FUNCTION_BLOCK

FUNCTION_BLOCK "Počítadlo"   // FB3, LAD
{ S7_Optimized_Access := 'FALSE' }
VERSION : 0.1
   VAR
      Linka1 : "Pocet";
      Linka2 : "Pocet";
      "Plná paleta D11" : Bool;
      "Plná paleta D12" : Bool;
   END_VAR
BEGIN

REGION Network 1
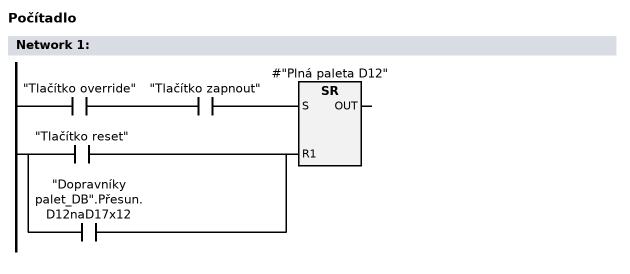
   RUNG wire#powerrail
      Contact( "Tlačítko override" )
      Contact( "Tlačítko zapnout" )
      S_SR(operand := #"Plná paleta D12", r1 := wire#w1)
   END_RUNG
   RUNG wire#powerrail
      Contact( "Tlačítko reset" )
   END_RUNG wire#w1
   RUNG wire#powerrail
      Contact( "Dopravníky palet_DB".Přesun.D12naD17x12 )
   END_RUNG wire#w1
   // the same network as SCL:
   IF "Tlačítko override" AND "Tlačítko zapnout" THEN
       #"Plná paleta D12" := TRUE;   // SR flip-flop
   END_IF;
   IF "Tlačítko reset" OR "Dopravníky palet_DB".Přesun.D12naD17x12 THEN #"Plná paleta D12" := FALSE; END_IF;
END_REGION
END_FUNCTION_BLOCK

FUNCTION_BLOCK "Pallet dispenser"   // FB4, LAD
{ S7_Optimized_Access := 'FALSE' }
VERSION : 0.1
   VAR_INPUT
      DOWN_accident : Bool;
      Dispenser_is_down : Bool;
      Dispenser_in_middle : Bool;
      Dispenser_is_up : Bool;
      UP_accident : Bool;
      Circuit_breaker : Bool;
      Arms_are_open : Bool;
      Arms_are_close : Bool;
      Pallet_under_dispenser : Bool;
      Automatic_mode : Bool;
      Power_circuit_OK : Bool;
      Pneumatic_OK : Bool;
      Sensor_before_dispenser : Bool;
      Button_Open_door : Bool;
      Sensor_door_are_open : Bool;
      Button_Door_are_close : Bool;
      OP_up : Bool;
      OP_down : Bool;
      OP_Airs_move : Bool;
      Pallet_transfare : Bool;
      Button_RESET : Bool;
      "Časovač 1" : Timer;
      "Časovač 2" : Timer;
      "Časovač 3" : Timer;
      "Časovač 4" : Timer;
      "Časovač 5" : Timer;
   END_VAR
   VAR_OUTPUT
      Let_go_UP : Bool;
      Let_go_DOWN : Bool;
      Break : Bool;
      Let_arms_close : Bool;
      Let_arms_open : Bool;
      Let_open_door : Bool;
      Led_door_are_open : Bool;
   END_VAR
   VAR
      Paleta_polozena : Bool;
      Stop_v_rucnim : Bool;
      Hrana_stop_v_rucnim : Bool;
      Pozadavek_otevreni_dveri : Bool;
      Door_opened : Bool;
      Arms_are_close_pozition : Bool;
   END_VAR
   VAR_TEMP   // added for the SCL form of the ladder/FBD networks
      _s5time1 : S5Time;
      _w1 : Bool;
   END_VAR
BEGIN

REGION Network 1
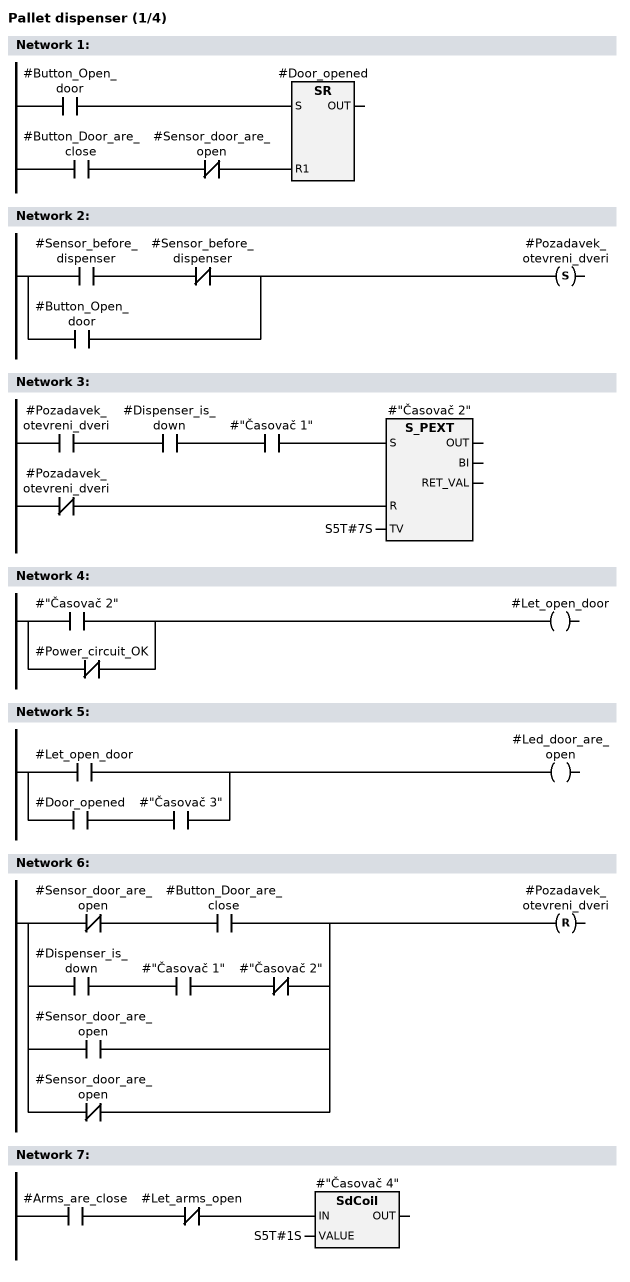
   RUNG wire#powerrail
      Contact( #Button_Open_door )
      S_SR(operand := #Door_opened, r1 := wire#w1)
   END_RUNG
   RUNG wire#powerrail
      Contact( #Button_Door_are_close )
      I_Contact( #Sensor_door_are_open )
   END_RUNG wire#w1
   // the same network as SCL:
   IF #Button_Open_door THEN
       #Door_opened := TRUE;   // SR flip-flop
   END_IF;
   IF #Button_Door_are_close AND NOT #Sensor_door_are_open THEN #Door_opened := FALSE; END_IF;
END_REGION

REGION Network 2
   RUNG wire#powerrail
      Contact( #Sensor_before_dispenser )
      I_Contact( #Sensor_before_dispenser )
      wire#w1
      S_Coil( #Pozadavek_otevreni_dveri )
   END_RUNG
   RUNG wire#powerrail
      Contact( #Button_Open_door )
   END_RUNG wire#w1
   // the same network as SCL:
   IF (#Sensor_before_dispenser AND NOT #Sensor_before_dispenser) OR #Button_Open_door THEN
       #Pozadavek_otevreni_dveri := TRUE;
   END_IF;
END_REGION

REGION Network 3
   RUNG wire#powerrail
      Contact( #Pozadavek_otevreni_dveri )
      Contact( #Dispenser_is_down )
      Contact( #"Časovač 1" )
      S_PEXT(T_NO := #"Časovač 2", R := wire#w1, TV := S5T#7S, BI =>, RET_VAL =>)
   END_RUNG
   RUNG wire#powerrail
      I_Contact( #Pozadavek_otevreni_dveri )
   END_RUNG wire#w1
   // the same network as SCL:
   #_s5time1 := S_PEXT(T_NO := #"Časovač 2",
                       S := #Pozadavek_otevreni_dveri AND #Dispenser_is_down AND #"Časovač 1",
                       R := NOT #Pozadavek_otevreni_dveri,
                       TV := S5T#7S);
END_REGION

REGION Network 4
   RUNG wire#powerrail
      Contact( #"Časovač 2" )
      wire#w1
      Coil( #Let_open_door )
   END_RUNG
   RUNG wire#powerrail
      I_Contact( #Power_circuit_OK )
   END_RUNG wire#w1
   // the same network as SCL:
   #Let_open_door := #"Časovač 2" OR NOT #Power_circuit_OK;
END_REGION

REGION Network 5
   RUNG wire#powerrail
      Contact( #Let_open_door )
      wire#w1
      Coil( #Led_door_are_open )
   END_RUNG
   RUNG wire#powerrail
      Contact( #Door_opened )
      Contact( #"Časovač 3" )
   END_RUNG wire#w1
   // the same network as SCL:
   #Led_door_are_open := #Let_open_door OR (#Door_opened AND #"Časovač 3");
END_REGION

REGION Network 6
   RUNG wire#powerrail
      I_Contact( #Sensor_door_are_open )
      Contact( #Button_Door_are_close )
      wire#w1
      R_Coil( #Pozadavek_otevreni_dveri )
   END_RUNG
   RUNG wire#powerrail
      Contact( #Dispenser_is_down )
      Contact( #"Časovač 1" )
      I_Contact( #"Časovač 2" )
   END_RUNG wire#w1
   RUNG wire#powerrail
      Contact( #Sensor_door_are_open )
   END_RUNG wire#w1
   RUNG wire#powerrail
      I_Contact( #Sensor_door_are_open )
   END_RUNG wire#w1
   // the same network as SCL:
   IF (NOT #Sensor_door_are_open AND #Button_Door_are_close) OR (#Dispenser_is_down AND #"Časovač 1" AND NOT #"Časovač 2") OR #Sensor_door_are_open OR NOT #Sensor_door_are_open THEN
       #Pozadavek_otevreni_dveri := FALSE;
   END_IF;
END_REGION

REGION Network 7
   // no SCL statement known for SdCoil: written as a call
   SdCoil(in := #Arms_are_close AND NOT #Let_arms_open, value := S5T#1S, operand := #"Časovač 4");
END_REGION

REGION Network 8
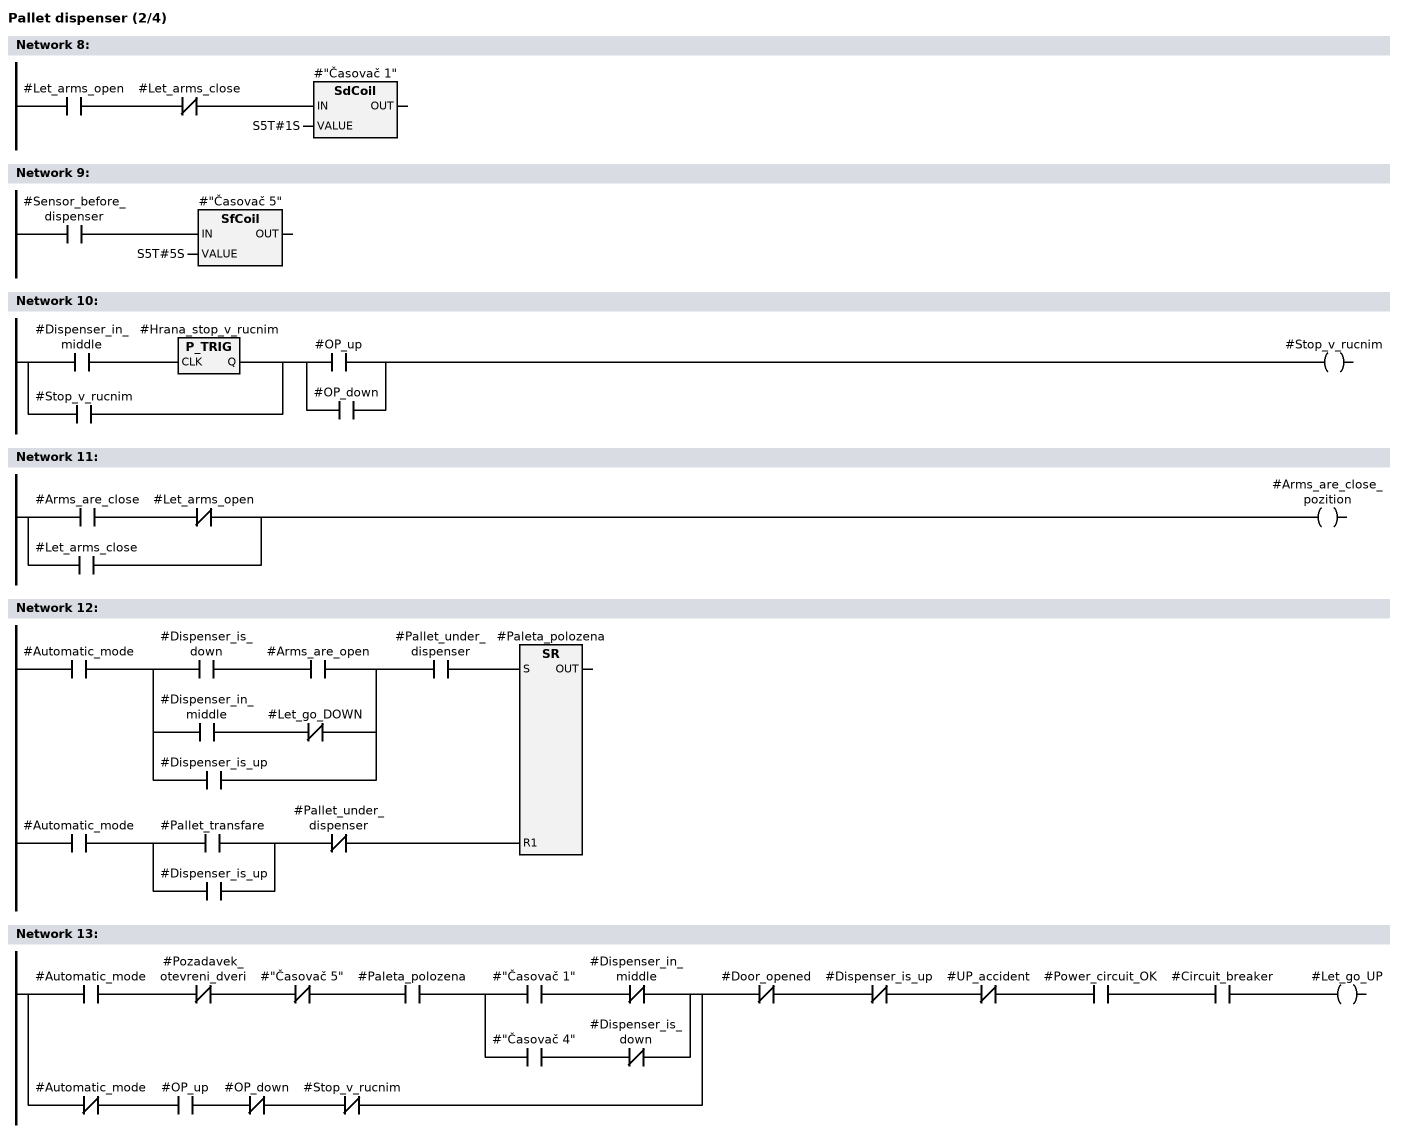
   // no SCL statement known for SdCoil: written as a call
   SdCoil(in := #Let_arms_open AND NOT #Let_arms_close, value := S5T#1S, operand := #"Časovač 1");
END_REGION

REGION Network 9
   // no SCL statement known for SfCoil: written as a call
   SfCoil(in := #Sensor_before_dispenser, value := S5T#5S, operand := #"Časovač 5");
END_REGION

REGION Network 10
   RUNG wire#powerrail
      Contact( #Dispenser_in_middle )
      P_Trig( #Hrana_stop_v_rucnim )
      wire#w1
      Contact( #OP_up )
      wire#w2
      Coil( #Stop_v_rucnim )
   END_RUNG
   RUNG wire#powerrail
      Contact( #Stop_v_rucnim )
   END_RUNG wire#w1
   RUNG wire#w1
      Contact( #OP_down )
   END_RUNG wire#w2
   // the same network as SCL:
   #_w1 := #Dispenser_in_middle AND NOT #Hrana_stop_v_rucnim;   // rising edge
   #Hrana_stop_v_rucnim := #Dispenser_in_middle;
   #Stop_v_rucnim := (#_w1 OR #Stop_v_rucnim) AND (#OP_up OR #OP_down);
END_REGION

REGION Network 11
   RUNG wire#powerrail
      Contact( #Arms_are_close )
      I_Contact( #Let_arms_open )
      wire#w1
      Coil( #Arms_are_close_pozition )
   END_RUNG
   RUNG wire#powerrail
      Contact( #Let_arms_close )
   END_RUNG wire#w1
   // the same network as SCL:
   #Arms_are_close_pozition := (#Arms_are_close AND NOT #Let_arms_open) OR #Let_arms_close;
END_REGION

REGION Network 12
   RUNG wire#powerrail
      Contact( #Automatic_mode )
      wire#w1
      Contact( #Dispenser_is_down )
      Contact( #Arms_are_open )
      wire#w2
      Contact( #Pallet_under_dispenser )
      S_SR(operand := #Paleta_polozena, r1 := wire#w5)
   END_RUNG
   RUNG wire#w1
      Contact( #Dispenser_in_middle )
      I_Contact( #Let_go_DOWN )
   END_RUNG wire#w2
   RUNG wire#w1
      Contact( #Dispenser_is_up )
   END_RUNG wire#w2
   RUNG wire#powerrail
      Contact( #Automatic_mode )
      wire#w3
      Contact( #Pallet_transfare )
      wire#w4
      I_Contact( #Pallet_under_dispenser )
   END_RUNG wire#w5
   RUNG wire#w3
      Contact( #Dispenser_is_up )
   END_RUNG wire#w4
   // the same network as SCL:
   IF #Automatic_mode AND ((#Dispenser_is_down AND #Arms_are_open) OR (#Dispenser_in_middle AND NOT #Let_go_DOWN) OR #Dispenser_is_up) AND #Pallet_under_dispenser THEN
       #Paleta_polozena := TRUE;   // SR flip-flop
   END_IF;
   IF #Automatic_mode AND (#Pallet_transfare OR #Dispenser_is_up) AND NOT #Pallet_under_dispenser THEN
       #Paleta_polozena := FALSE;
   END_IF;
END_REGION

REGION Network 13
   RUNG wire#powerrail
      Contact( #Automatic_mode )
      I_Contact( #Pozadavek_otevreni_dveri )
      I_Contact( #"Časovač 5" )
      Contact( #Paleta_polozena )
      wire#w1
      Contact( #"Časovač 1" )
      I_Contact( #Dispenser_in_middle )
      wire#w2
      I_Contact( #Door_opened )
      I_Contact( #Dispenser_is_up )
      I_Contact( #UP_accident )
      Contact( #Power_circuit_OK )
      Contact( #Circuit_breaker )
      Coil( #Let_go_UP )
   END_RUNG
   RUNG wire#w1
      Contact( #"Časovač 4" )
      I_Contact( #Dispenser_is_down )
   END_RUNG wire#w2
   RUNG wire#powerrail
      I_Contact( #Automatic_mode )
      Contact( #OP_up )
      I_Contact( #OP_down )
      I_Contact( #Stop_v_rucnim )
   END_RUNG wire#w2
   // the same network as SCL:
   #Let_go_UP := ((#Automatic_mode AND NOT #Pozadavek_otevreni_dveri AND NOT #"Časovač 5" AND #Paleta_polozena AND ((#"Časovač 1" AND NOT #Dispenser_in_middle) OR (#"Časovač 4" AND NOT #Dispenser_is_down))) OR (NOT #Automatic_mode AND #OP_up AND NOT #OP_down AND NOT #Stop_v_rucnim)) AND NOT #Door_opened AND NOT #Dispenser_is_up AND NOT #UP_accident AND #Power_circuit_OK AND #Circuit_breaker;
END_REGION

REGION Network 14
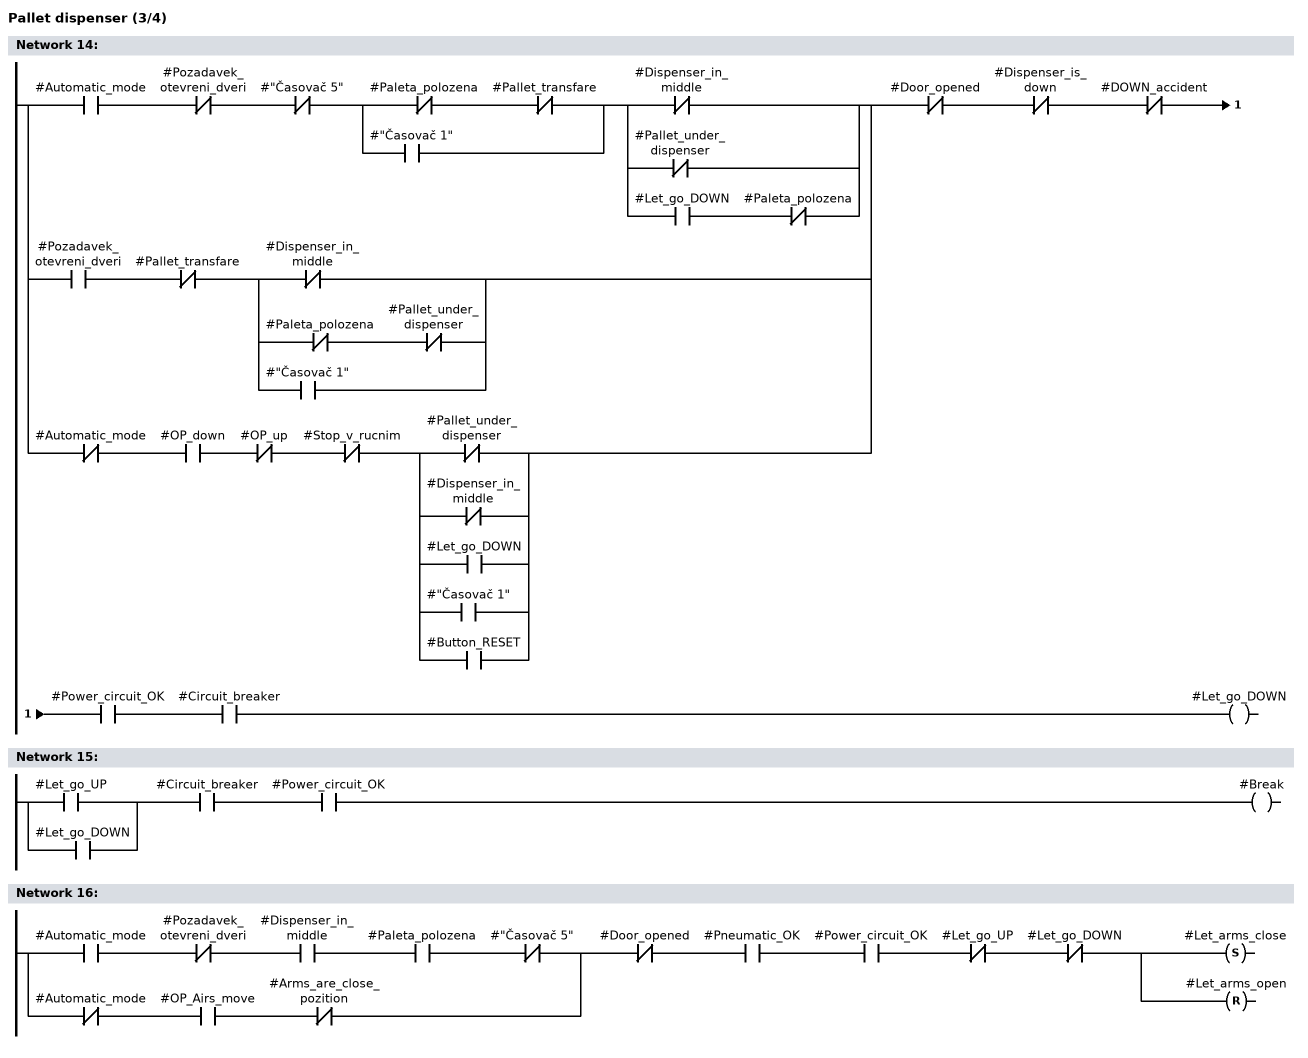
   RUNG wire#powerrail
      Contact( #Automatic_mode )
      I_Contact( #Pozadavek_otevreni_dveri )
      I_Contact( #"Časovač 5" )
      wire#w1
      I_Contact( #Paleta_polozena )
      I_Contact( #Pallet_transfare )
      wire#w2
      I_Contact( #Dispenser_in_middle )
      wire#w3
      I_Contact( #Door_opened )
      I_Contact( #Dispenser_is_down )
      I_Contact( #DOWN_accident )
      Contact( #Power_circuit_OK )
      Contact( #Circuit_breaker )
      Coil( #Let_go_DOWN )
   END_RUNG
   RUNG wire#w1
      Contact( #"Časovač 1" )
   END_RUNG wire#w2
   RUNG wire#w2
      I_Contact( #Pallet_under_dispenser )
   END_RUNG wire#w3
   RUNG wire#w2
      Contact( #Let_go_DOWN )
      I_Contact( #Paleta_polozena )
   END_RUNG wire#w3
   RUNG wire#powerrail
      Contact( #Pozadavek_otevreni_dveri )
      I_Contact( #Pallet_transfare )
      wire#w4
      I_Contact( #Dispenser_in_middle )
   END_RUNG wire#w3
   RUNG wire#w4
      I_Contact( #Paleta_polozena )
      I_Contact( #Pallet_under_dispenser )
   END_RUNG wire#w3
   RUNG wire#w4
      Contact( #"Časovač 1" )
   END_RUNG wire#w3
   RUNG wire#powerrail
      I_Contact( #Automatic_mode )
      Contact( #OP_down )
      I_Contact( #OP_up )
      I_Contact( #Stop_v_rucnim )
      wire#w5
      I_Contact( #Pallet_under_dispenser )
   END_RUNG wire#w3
   RUNG wire#w5
      I_Contact( #Dispenser_in_middle )
   END_RUNG wire#w3
   RUNG wire#w5
      Contact( #Let_go_DOWN )
   END_RUNG wire#w3
   RUNG wire#w5
      Contact( #"Časovač 1" )
   END_RUNG wire#w3
   RUNG wire#w5
      Contact( #Button_RESET )
   END_RUNG wire#w3
   // the same network as SCL:
   #Let_go_DOWN := ((#Automatic_mode AND NOT #Pozadavek_otevreni_dveri AND NOT #"Časovač 5" AND ((NOT #Paleta_polozena AND NOT #Pallet_transfare) OR #"Časovač 1") AND (NOT #Dispenser_in_middle OR NOT #Pallet_under_dispenser OR (#Let_go_DOWN AND NOT #Paleta_polozena))) OR (#Pozadavek_otevreni_dveri AND NOT #Pallet_transfare AND (NOT #Dispenser_in_middle OR (NOT #Paleta_polozena AND NOT #Pallet_under_dispenser) OR #"Časovač 1")) OR (NOT #Automatic_mode AND #OP_down AND NOT #OP_up AND NOT #Stop_v_rucnim AND (NOT #Pallet_under_dispenser OR NOT #Dispenser_in_middle OR #Let_go_DOWN OR #"Časovač 1" OR #Button_RESET))) AND NOT #Door_opened AND NOT #Dispenser_is_down AND NOT #DOWN_accident AND #Power_circuit_OK AND #Circuit_breaker;
END_REGION

REGION Network 15
   RUNG wire#powerrail
      Contact( #Let_go_UP )
      wire#w1
      Contact( #Circuit_breaker )
      Contact( #Power_circuit_OK )
      Coil( #Break )
   END_RUNG
   RUNG wire#powerrail
      Contact( #Let_go_DOWN )
   END_RUNG wire#w1
   // the same network as SCL:
   #Break := (#Let_go_UP OR #Let_go_DOWN) AND #Circuit_breaker AND #Power_circuit_OK;
END_REGION

REGION Network 16
   RUNG wire#powerrail
      Contact( #Automatic_mode )
      I_Contact( #Pozadavek_otevreni_dveri )
      Contact( #Dispenser_in_middle )
      Contact( #Paleta_polozena )
      I_Contact( #"Časovač 5" )
      wire#w1
      I_Contact( #Door_opened )
      Contact( #Pneumatic_OK )
      Contact( #Power_circuit_OK )
      I_Contact( #Let_go_UP )
      I_Contact( #Let_go_DOWN )
      wire#w2
      S_Coil( #Let_arms_close )
   END_RUNG
   RUNG wire#powerrail
      I_Contact( #Automatic_mode )
      Contact( #OP_Airs_move )
      I_Contact( #Arms_are_close_pozition )
   END_RUNG wire#w1
   RUNG wire#w2
      R_Coil( #Let_arms_open )
   END_RUNG
   // the same network as SCL:
   IF ((#Automatic_mode AND NOT #Pozadavek_otevreni_dveri AND #Dispenser_in_middle AND #Paleta_polozena AND NOT #"Časovač 5") OR (NOT #Automatic_mode AND #OP_Airs_move AND NOT #Arms_are_close_pozition)) AND NOT #Door_opened AND #Pneumatic_OK AND #Power_circuit_OK AND NOT #Let_go_UP AND NOT #Let_go_DOWN THEN
       #Let_arms_close := TRUE;
       #Let_arms_open := FALSE;
   END_IF;
END_REGION

REGION Network 17
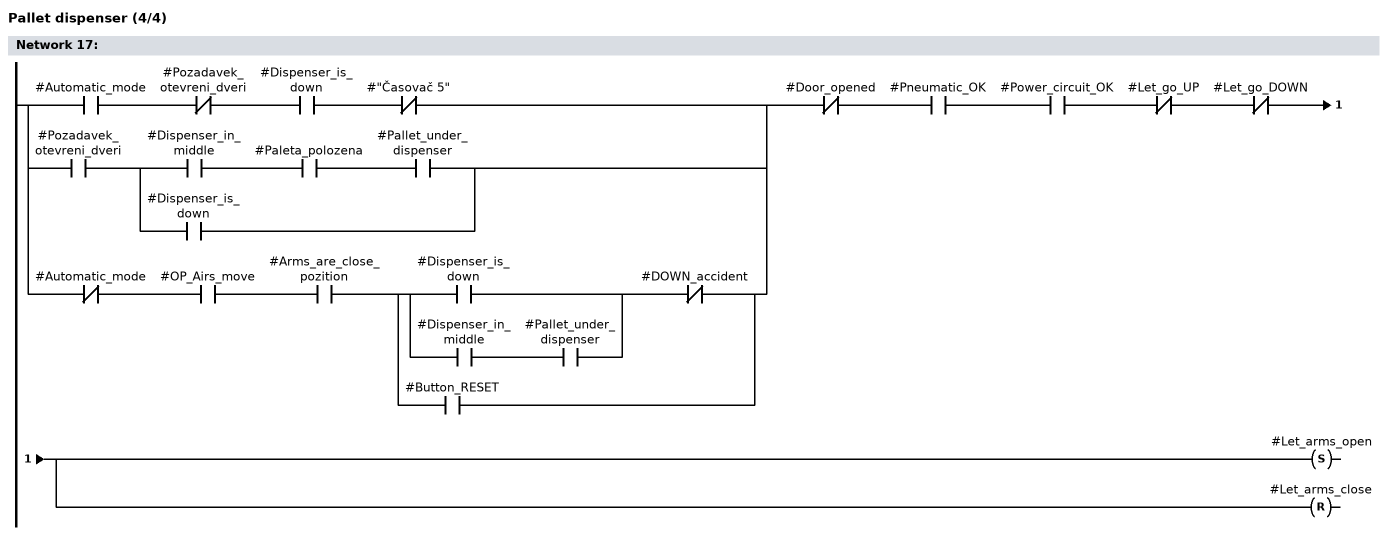
   RUNG wire#powerrail
      Contact( #Automatic_mode )
      I_Contact( #Pozadavek_otevreni_dveri )
      Contact( #Dispenser_is_down )
      I_Contact( #"Časovač 5" )
      wire#w1
      I_Contact( #Door_opened )
      Contact( #Pneumatic_OK )
      Contact( #Power_circuit_OK )
      I_Contact( #Let_go_UP )
      I_Contact( #Let_go_DOWN )
      wire#w5
      S_Coil( #Let_arms_open )
   END_RUNG
   RUNG wire#powerrail
      Contact( #Pozadavek_otevreni_dveri )
      wire#w2
      Contact( #Dispenser_in_middle )
      Contact( #Paleta_polozena )
      Contact( #Pallet_under_dispenser )
   END_RUNG wire#w1
   RUNG wire#w2
      Contact( #Dispenser_is_down )
   END_RUNG wire#w1
   RUNG wire#powerrail
      I_Contact( #Automatic_mode )
      Contact( #OP_Airs_move )
      Contact( #Arms_are_close_pozition )
      wire#w3
      Contact( #Dispenser_is_down )
      wire#w4
      I_Contact( #DOWN_accident )
   END_RUNG wire#w1
   RUNG wire#w3
      Contact( #Dispenser_in_middle )
      Contact( #Pallet_under_dispenser )
   END_RUNG wire#w4
   RUNG wire#w3
      Contact( #Button_RESET )
   END_RUNG wire#w1
   RUNG wire#w5
      R_Coil( #Let_arms_close )
   END_RUNG
   // the same network as SCL:
   IF ((#Automatic_mode AND NOT #Pozadavek_otevreni_dveri AND #Dispenser_is_down AND NOT #"Časovač 5") OR (#Pozadavek_otevreni_dveri AND ((#Dispenser_in_middle AND #Paleta_polozena AND #Pallet_under_dispenser) OR #Dispenser_is_down)) OR (NOT #Automatic_mode AND #OP_Airs_move AND #Arms_are_close_pozition AND (((#Dispenser_is_down OR (#Dispenser_in_middle AND #Pallet_under_dispenser)) AND NOT #DOWN_accident) OR #Button_RESET))) AND NOT #Door_opened AND #Pneumatic_OK AND #Power_circuit_OK AND NOT #Let_go_UP AND NOT #Let_go_DOWN THEN
       #Let_arms_open := TRUE;
       #Let_arms_close := FALSE;
   END_IF;
END_REGION
END_FUNCTION_BLOCK

FUNCTION_BLOCK "Dopravníky kartonů linka 1"   // FB5, LAD
{ S7_Optimized_Access := 'FALSE' }
VERSION : 0.1
   VAR
      PočetNaP49 : Int;
      PlnáŘadaD49 : Bool;
      "Srovnaná řada na D49" : Bool;
      PHranaT40 : Bool;
      "P35 Odjezd volný" : Bool;
      "P35 Nájezd kartonů" : Bool;
      "P35 Hrana nájezdu" : Bool;
      "P35 Nájezd na pozici" : Bool;
      "P35 zpomalení" : Bool;
      "Karton na počítání" : Bool;
   END_VAR
   VAR_TEMP
      Dummy : Bool;
      "Klapka P47.2 nahoru" : Bool;
      "Klapka P47.2 dolů" : Bool;
      "Klapka P47.1 nahoru" : Bool;
      "Klapka P47.1 dolů" : Bool;
      "Klapka P33 nahoru" : Bool;
      "Klapka P33 dolů" : Bool;
   END_VAR
   VAR_TEMP   // added for the SCL form of the ladder/FBD networks
      _w1 : Bool;
      _s5time1 : S5Time;
      _w2 : Bool;
      _s5time2 : S5Time;
      _w3 : Bool;
   END_VAR
BEGIN

REGION Network 1
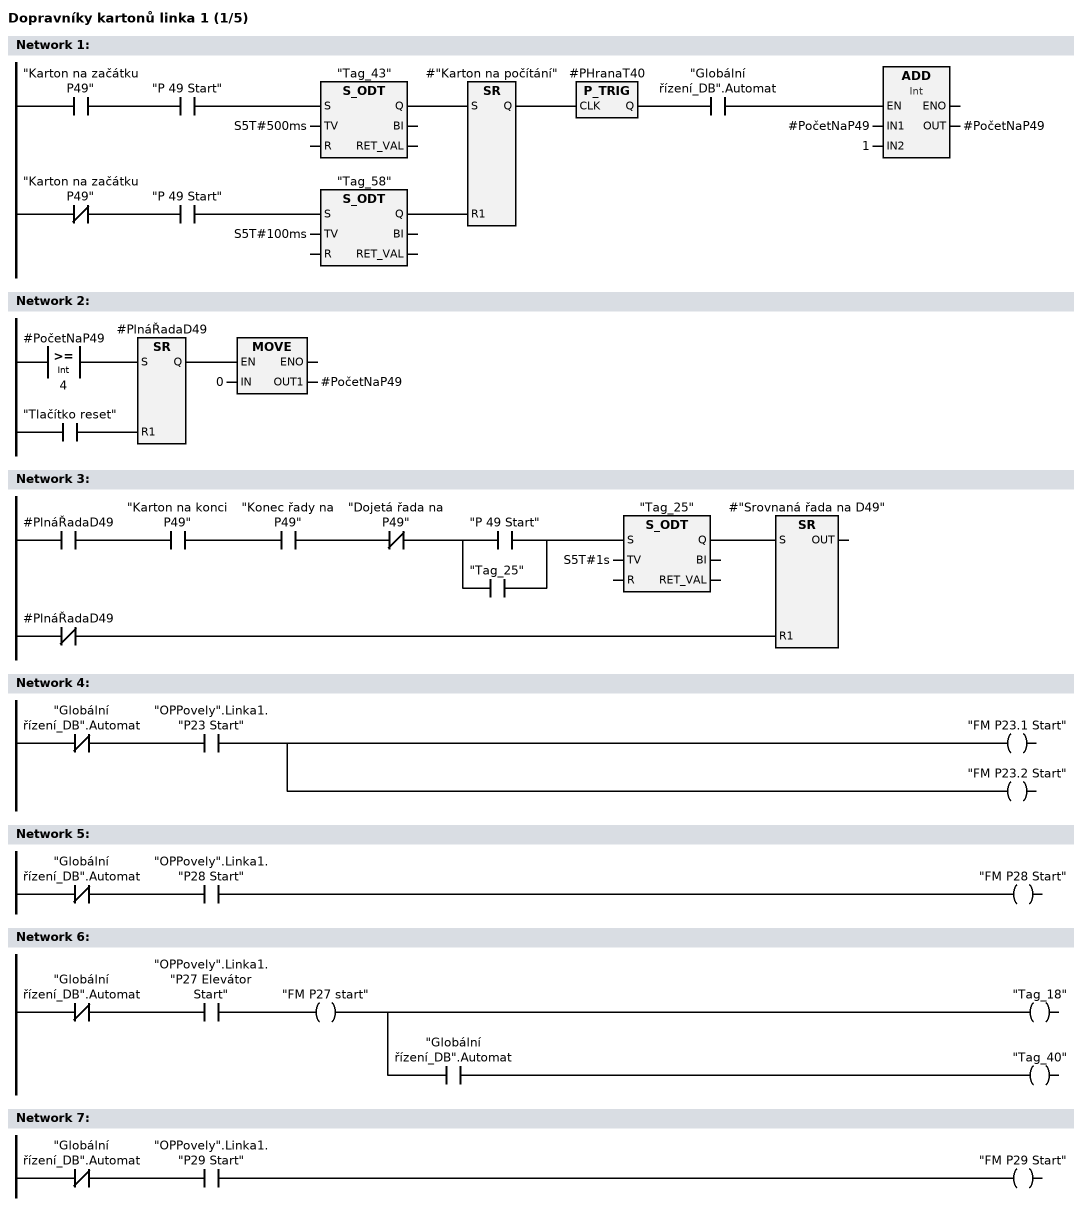
   RUNG wire#powerrail
      Contact( "Karton na začátku P49" )
      Contact( "P 49 Start" )
      S_ODT(T_NO := "Tag_43", TV := S5T#500ms, R :=, BI =>, RET_VAL =>)
      S_SR(operand := #"Karton na počítání", r1 := wire#w1)
      P_Trig( #PHranaT40 )
      Contact( "Globální řízení_DB".Automat )
      { S7_Templates := "SrcType := Int"; S7_GenerateENO := "TRUE" } Add(in1 := #PočetNaP49, in2 := 1, out => #PočetNaP49)
   END_RUNG
   RUNG wire#powerrail
      I_Contact( "Karton na začátku P49" )
      Contact( "P 49 Start" )
      S_ODT(T_NO := "Tag_58", TV := S5T#100ms, R :=, BI =>, RET_VAL =>)
   END_RUNG wire#w1
   // the same network as SCL:
   #_s5time1 := S_ODT(T_NO := "Tag_43",
                      S := "Karton na začátku P49" AND "P 49 Start",
                      TV := S5T#500ms,
                      Q => #_w1);
   #_s5time2 := S_ODT(T_NO := "Tag_58",
                      S := NOT "Karton na začátku P49" AND "P 49 Start",
                      TV := S5T#100ms,
                      Q => #_w2);
   IF #_w1 THEN
       #"Karton na počítání" := TRUE;   // SR flip-flop
   END_IF;
   IF #_w2 THEN #"Karton na počítání" := FALSE; END_IF;
   #_w3 := #"Karton na počítání" AND NOT #PHranaT40;   // rising edge
   #PHranaT40 := #"Karton na počítání";
   IF #_w3 AND "Globální řízení_DB".Automat THEN #PočetNaP49 := #PočetNaP49 + 1; END_IF;
END_REGION

REGION Network 2
   RUNG wire#powerrail
      { S7_Templates := "SrcType := Int" } GE_Contact(in1 := #PočetNaP49, in2 := 4)
      S_SR(operand := #PlnáŘadaD49, r1 := wire#w1)
      { S7_GenerateENO := "TRUE" } Move(in := 0, out1 => #PočetNaP49)
   END_RUNG
   RUNG wire#powerrail
      Contact( "Tlačítko reset" )
   END_RUNG wire#w1
   // the same network as SCL:
   IF #PočetNaP49 >= 4 THEN
       #PlnáŘadaD49 := TRUE;   // SR flip-flop
   END_IF;
   IF "Tlačítko reset" THEN #PlnáŘadaD49 := FALSE; END_IF;
   IF #PlnáŘadaD49 THEN #PočetNaP49 := 0; END_IF;
END_REGION

REGION Network 3
   RUNG wire#powerrail
      Contact( #PlnáŘadaD49 )
      Contact( "Karton na konci P49" )
      Contact( "Konec řady na P49" )
      I_Contact( "Dojetá řada na P49" )
      wire#w1
      Contact( "P 49 Start" )
      wire#w2
      S_ODT(T_NO := "Tag_25", TV := S5T#1s, R :=, BI =>, RET_VAL =>)
      S_SR(operand := #"Srovnaná řada na D49", r1 := wire#w3)
   END_RUNG
   RUNG wire#w1
      Contact( "Tag_25" )
   END_RUNG wire#w2
   RUNG wire#powerrail
      I_Contact( #PlnáŘadaD49 )
   END_RUNG wire#w3
   // the same network as SCL:
   #_s5time1 := S_ODT(T_NO := "Tag_25",
                      S := #PlnáŘadaD49 AND "Karton na konci P49" AND "Konec řady na P49" AND NOT "Dojetá řada na P49" AND ("P 49 Start" OR "Tag_25"),
                      TV := S5T#1s,
                      Q => #_w1);
   IF #_w1 THEN
       #"Srovnaná řada na D49" := TRUE;   // SR flip-flop
   END_IF;
   IF NOT #PlnáŘadaD49 THEN #"Srovnaná řada na D49" := FALSE; END_IF;
END_REGION

REGION Network 4
   RUNG wire#powerrail
      I_Contact( "Globální řízení_DB".Automat )
      Contact( "OPPovely".Linka1."P23 Start" )
      wire#w1
      Coil( "FM P23.1 Start" )
   END_RUNG
   RUNG wire#w1
      Coil( "FM P23.2 Start" )
   END_RUNG
   // the same network as SCL:
   "FM P23.1 Start" := NOT "Globální řízení_DB".Automat AND "OPPovely".Linka1."P23 Start";
   "FM P23.2 Start" := "FM P23.1 Start";
END_REGION

REGION Network 5
   RUNG wire#powerrail
      I_Contact( "Globální řízení_DB".Automat )
      Contact( "OPPovely".Linka1."P28 Start" )
      Coil( "FM P28 Start" )
   END_RUNG
   // the same network as SCL:
   "FM P28 Start" := NOT "Globální řízení_DB".Automat AND "OPPovely".Linka1."P28 Start";
END_REGION

REGION Network 6
   RUNG wire#powerrail
      I_Contact( "Globální řízení_DB".Automat )
      Contact( "OPPovely".Linka1."P27 Elevátor Start" )
      Coil( "FM P27 start" )
      wire#w1
      Coil( "Tag_18" )
   END_RUNG
   RUNG wire#w1
      Contact( "Globální řízení_DB".Automat )
      Coil( "Tag_40" )
   END_RUNG
   // the same network as SCL:
   "FM P27 start" := NOT "Globální řízení_DB".Automat AND "OPPovely".Linka1."P27 Elevátor Start";
   "Tag_18" := "FM P27 start";
   "Tag_40" := "FM P27 start" AND "Globální řízení_DB".Automat;
END_REGION

REGION Network 7
   RUNG wire#powerrail
      I_Contact( "Globální řízení_DB".Automat )
      Contact( "OPPovely".Linka1."P29 Start" )
      Coil( "FM P29 Start" )
   END_RUNG
   // the same network as SCL:
   "FM P29 Start" := NOT "Globální řízení_DB".Automat AND "OPPovely".Linka1."P29 Start";
END_REGION

REGION Network 9
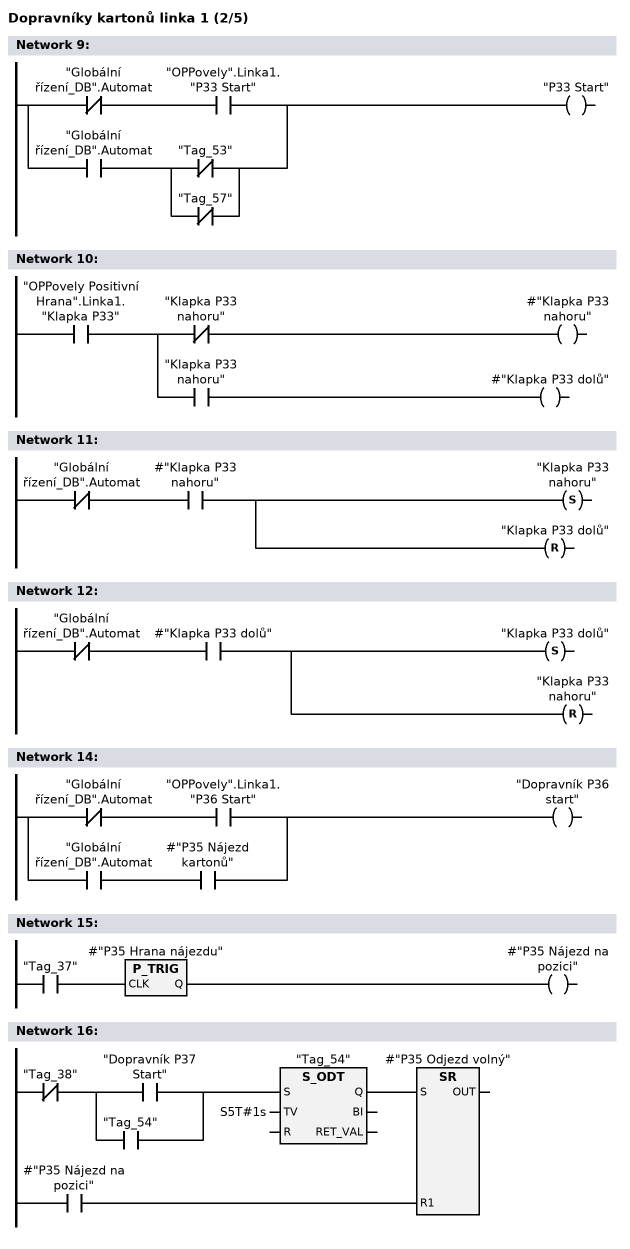
   RUNG wire#powerrail
      I_Contact( "Globální řízení_DB".Automat )
      Contact( "OPPovely".Linka1."P33 Start" )
      wire#w1
      Coil( "P33 Start" )
   END_RUNG
   RUNG wire#powerrail
      Contact( "Globální řízení_DB".Automat )
      wire#w2
      I_Contact( "Tag_53" )
   END_RUNG wire#w1
   RUNG wire#w2
      I_Contact( "Tag_57" )
   END_RUNG wire#w1
   // the same network as SCL:
   "P33 Start" := (NOT "Globální řízení_DB".Automat AND "OPPovely".Linka1."P33 Start") OR ("Globální řízení_DB".Automat AND (NOT "Tag_53" OR NOT "Tag_57"));
END_REGION

REGION Network 10
   RUNG wire#powerrail
      Contact( "OPPovely Positivní Hrana".Linka1."Klapka P33" )
      wire#w1
      I_Contact( "Klapka P33 nahoru" )
      Coil( #"Klapka P33 nahoru" )
   END_RUNG
   RUNG wire#w1
      Contact( "Klapka P33 nahoru" )
      Coil( #"Klapka P33 dolů" )
   END_RUNG
   // the same network as SCL:
   #"Klapka P33 nahoru" := "OPPovely Positivní Hrana".Linka1."Klapka P33" AND NOT "Klapka P33 nahoru";
   #"Klapka P33 dolů" := "OPPovely Positivní Hrana".Linka1."Klapka P33" AND "Klapka P33 nahoru";
END_REGION

REGION Network 11
   RUNG wire#powerrail
      I_Contact( "Globální řízení_DB".Automat )
      Contact( #"Klapka P33 nahoru" )
      wire#w1
      S_Coil( "Klapka P33 nahoru" )
   END_RUNG
   RUNG wire#w1
      R_Coil( "Klapka P33 dolů" )
   END_RUNG
   // the same network as SCL:
   IF NOT "Globální řízení_DB".Automat AND #"Klapka P33 nahoru" THEN
       "Klapka P33 nahoru" := TRUE;
       "Klapka P33 dolů" := FALSE;
   END_IF;
END_REGION

REGION Network 12
   RUNG wire#powerrail
      I_Contact( "Globální řízení_DB".Automat )
      Contact( #"Klapka P33 dolů" )
      wire#w1
      S_Coil( "Klapka P33 dolů" )
   END_RUNG
   RUNG wire#w1
      R_Coil( "Klapka P33 nahoru" )
   END_RUNG
   // the same network as SCL:
   IF NOT "Globální řízení_DB".Automat AND #"Klapka P33 dolů" THEN
       "Klapka P33 dolů" := TRUE;
       "Klapka P33 nahoru" := FALSE;
   END_IF;
END_REGION

REGION Network 14
   RUNG wire#powerrail
      I_Contact( "Globální řízení_DB".Automat )
      Contact( "OPPovely".Linka1."P36 Start" )
      wire#w1
      Coil( "Dopravník P36 start" )
   END_RUNG
   RUNG wire#powerrail
      Contact( "Globální řízení_DB".Automat )
      Contact( #"P35 Nájezd kartonů" )
   END_RUNG wire#w1
   // the same network as SCL:
   "Dopravník P36 start" := (NOT "Globální řízení_DB".Automat AND "OPPovely".Linka1."P36 Start") OR ("Globální řízení_DB".Automat AND #"P35 Nájezd kartonů");
END_REGION

REGION Network 15
   RUNG wire#powerrail
      Contact( "Tag_37" )
      P_Trig( #"P35 Hrana nájezdu" )
      Coil( #"P35 Nájezd na pozici" )
   END_RUNG
   // the same network as SCL:
   #_w1 := "Tag_37" AND NOT #"P35 Hrana nájezdu";   // rising edge
   #"P35 Hrana nájezdu" := "Tag_37";
   #"P35 Nájezd na pozici" := #_w1;
END_REGION

REGION Network 16
   RUNG wire#powerrail
      I_Contact( "Tag_38" )
      wire#w1
      Contact( "Dopravník P37 Start" )
      wire#w2
      S_ODT(T_NO := "Tag_54", TV := S5T#1s, R :=, BI =>, RET_VAL =>)
      S_SR(operand := #"P35 Odjezd volný", r1 := wire#w3)
   END_RUNG
   RUNG wire#w1
      Contact( "Tag_54" )
   END_RUNG wire#w2
   RUNG wire#powerrail
      Contact( #"P35 Nájezd na pozici" )
   END_RUNG wire#w3
   // the same network as SCL:
   #_s5time1 := S_ODT(T_NO := "Tag_54",
                      S := NOT "Tag_38" AND ("Dopravník P37 Start" OR "Tag_54"),
                      TV := S5T#1s,
                      Q => #_w1);
   IF #_w1 THEN
       #"P35 Odjezd volný" := TRUE;   // SR flip-flop
   END_IF;
   IF #"P35 Nájezd na pozici" THEN #"P35 Odjezd volný" := FALSE; END_IF;
END_REGION

REGION Network 17
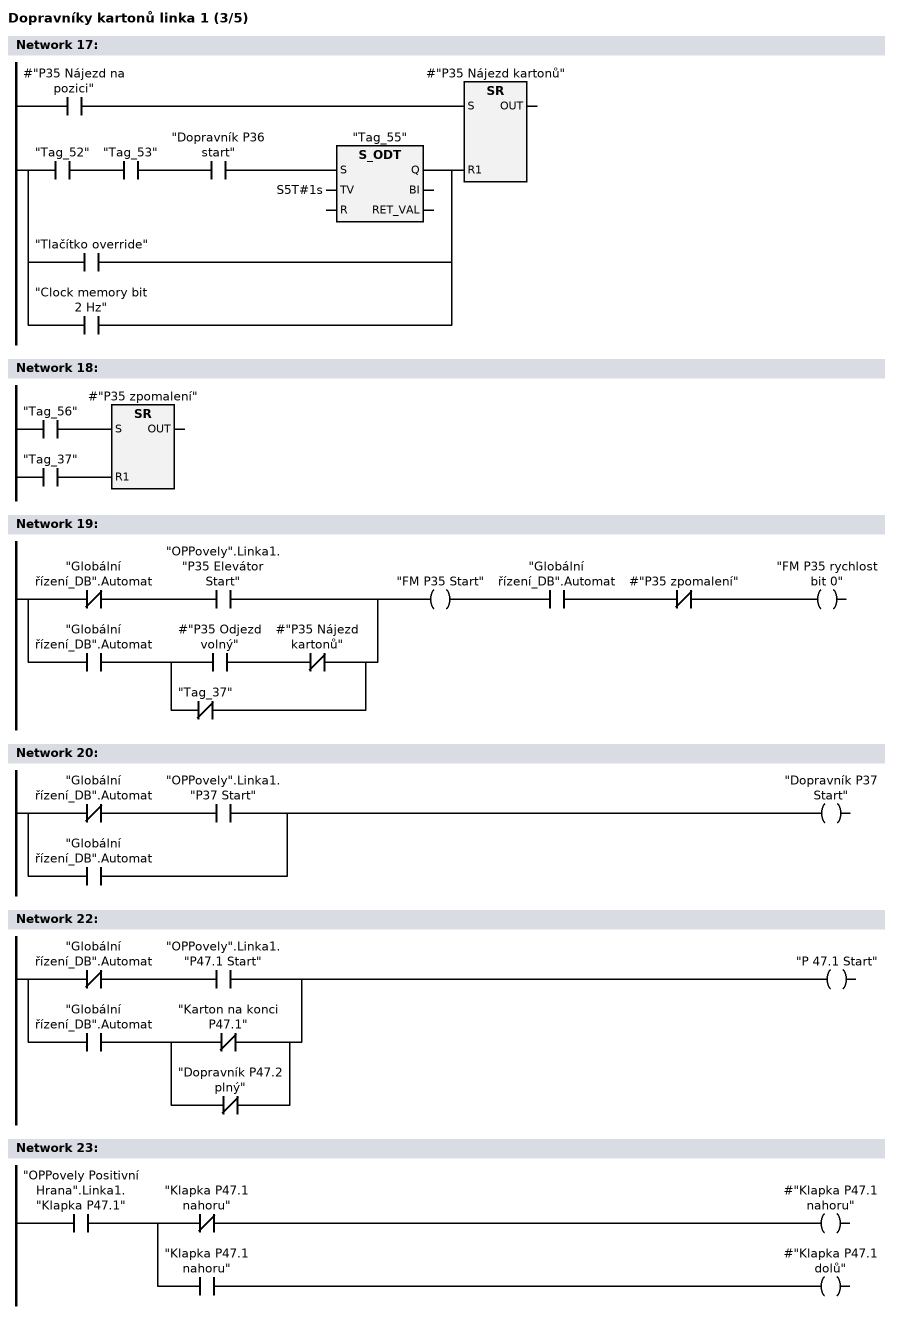
   RUNG wire#powerrail
      Contact( #"P35 Nájezd na pozici" )
      S_SR(operand := #"P35 Nájezd kartonů", r1 := wire#w1)
   END_RUNG
   RUNG wire#powerrail
      Contact( "Tag_52" )
      Contact( "Tag_53" )
      Contact( "Dopravník P36 start" )
      S_ODT(T_NO := "Tag_55", TV := S5T#1s, R :=, BI =>, RET_VAL =>)
   END_RUNG wire#w1
   RUNG wire#powerrail
      Contact( "Tlačítko override" )
   END_RUNG wire#w1
   RUNG wire#powerrail
      Contact( "Clock memory bit 2 Hz" )
   END_RUNG wire#w1
   // the same network as SCL:
   #_s5time1 := S_ODT(T_NO := "Tag_55",
                      S := "Tag_52" AND "Tag_53" AND "Dopravník P36 start",
                      TV := S5T#1s,
                      Q => #_w1);
   IF #"P35 Nájezd na pozici" THEN
       #"P35 Nájezd kartonů" := TRUE;   // SR flip-flop
   END_IF;
   IF #_w1 OR "Tlačítko override" OR "Clock memory bit 2 Hz" THEN #"P35 Nájezd kartonů" := FALSE; END_IF;
END_REGION

REGION Network 18
   RUNG wire#powerrail
      Contact( "Tag_56" )
      S_SR(operand := #"P35 zpomalení", r1 := wire#w1)
   END_RUNG
   RUNG wire#powerrail
      Contact( "Tag_37" )
   END_RUNG wire#w1
   // the same network as SCL:
   IF "Tag_56" THEN
       #"P35 zpomalení" := TRUE;   // SR flip-flop
   END_IF;
   IF "Tag_37" THEN #"P35 zpomalení" := FALSE; END_IF;
END_REGION

REGION Network 19
   RUNG wire#powerrail
      I_Contact( "Globální řízení_DB".Automat )
      Contact( "OPPovely".Linka1."P35 Elevátor Start" )
      wire#w1
      Coil( "FM P35 Start" )
      Contact( "Globální řízení_DB".Automat )
      I_Contact( #"P35 zpomalení" )
      Coil( "FM P35 rychlost bit 0" )
   END_RUNG
   RUNG wire#powerrail
      Contact( "Globální řízení_DB".Automat )
      wire#w2
      Contact( #"P35 Odjezd volný" )
      I_Contact( #"P35 Nájezd kartonů" )
   END_RUNG wire#w1
   RUNG wire#w2
      I_Contact( "Tag_37" )
   END_RUNG wire#w1
   // the same network as SCL:
   "FM P35 Start" := (NOT "Globální řízení_DB".Automat AND "OPPovely".Linka1."P35 Elevátor Start") OR ("Globální řízení_DB".Automat AND ((#"P35 Odjezd volný" AND NOT #"P35 Nájezd kartonů") OR NOT "Tag_37"));
   "FM P35 rychlost bit 0" := "FM P35 Start" AND "Globální řízení_DB".Automat AND NOT #"P35 zpomalení";
END_REGION

REGION Network 20
   RUNG wire#powerrail
      I_Contact( "Globální řízení_DB".Automat )
      Contact( "OPPovely".Linka1."P37 Start" )
      wire#w1
      Coil( "Dopravník P37 Start" )
   END_RUNG
   RUNG wire#powerrail
      Contact( "Globální řízení_DB".Automat )
   END_RUNG wire#w1
   // the same network as SCL:
   "Dopravník P37 Start" := (NOT "Globální řízení_DB".Automat AND "OPPovely".Linka1."P37 Start") OR "Globální řízení_DB".Automat;
END_REGION

REGION Network 22
   RUNG wire#powerrail
      I_Contact( "Globální řízení_DB".Automat )
      Contact( "OPPovely".Linka1."P47.1 Start" )
      wire#w1
      Coil( "P 47.1 Start" )
   END_RUNG
   RUNG wire#powerrail
      Contact( "Globální řízení_DB".Automat )
      wire#w2
      I_Contact( "Karton na konci P47.1" )
   END_RUNG wire#w1
   RUNG wire#w2
      I_Contact( "Dopravník P47.2 plný" )
   END_RUNG wire#w1
   // the same network as SCL:
   "P 47.1 Start" := (NOT "Globální řízení_DB".Automat AND "OPPovely".Linka1."P47.1 Start") OR ("Globální řízení_DB".Automat AND (NOT "Karton na konci P47.1" OR NOT "Dopravník P47.2 plný"));
END_REGION

REGION Network 23
   RUNG wire#powerrail
      Contact( "OPPovely Positivní Hrana".Linka1."Klapka P47.1" )
      wire#w1
      I_Contact( "Klapka P47.1 nahoru" )
      Coil( #"Klapka P47.1 nahoru" )
   END_RUNG
   RUNG wire#w1
      Contact( "Klapka P47.1 nahoru" )
      Coil( #"Klapka P47.1 dolů" )
   END_RUNG
   // the same network as SCL:
   #"Klapka P47.1 nahoru" := "OPPovely Positivní Hrana".Linka1."Klapka P47.1" AND NOT "Klapka P47.1 nahoru";
   #"Klapka P47.1 dolů" := "OPPovely Positivní Hrana".Linka1."Klapka P47.1" AND "Klapka P47.1 nahoru";
END_REGION

REGION Network 24
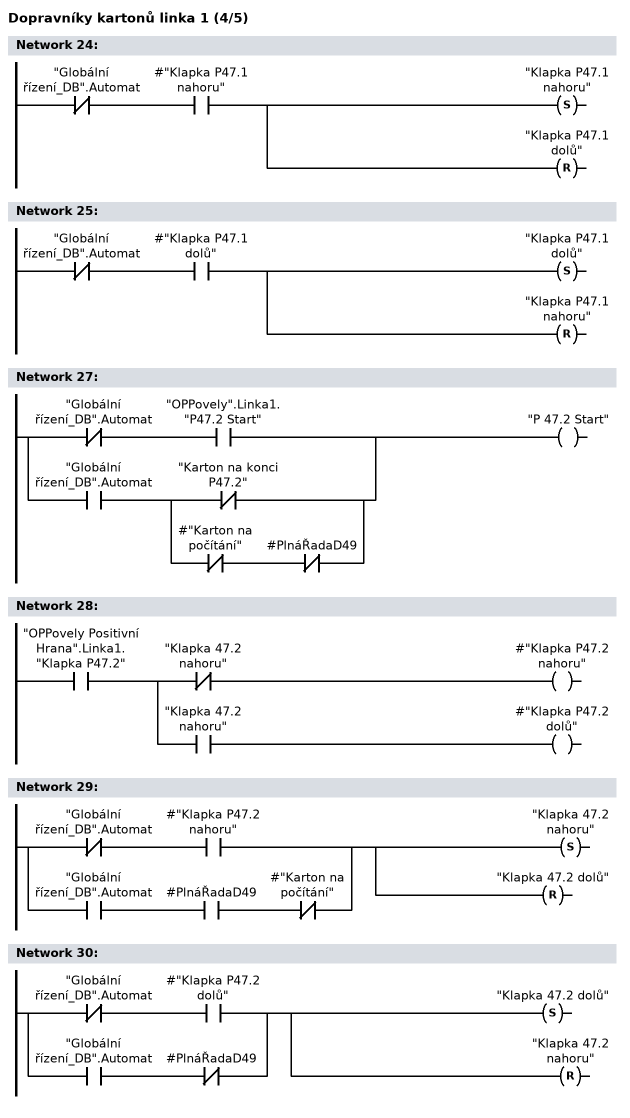
   RUNG wire#powerrail
      I_Contact( "Globální řízení_DB".Automat )
      Contact( #"Klapka P47.1 nahoru" )
      wire#w1
      S_Coil( "Klapka P47.1 nahoru" )
   END_RUNG
   RUNG wire#w1
      R_Coil( "Klapka P47.1 dolů" )
   END_RUNG
   // the same network as SCL:
   IF NOT "Globální řízení_DB".Automat AND #"Klapka P47.1 nahoru" THEN
       "Klapka P47.1 nahoru" := TRUE;
       "Klapka P47.1 dolů" := FALSE;
   END_IF;
END_REGION

REGION Network 25
   RUNG wire#powerrail
      I_Contact( "Globální řízení_DB".Automat )
      Contact( #"Klapka P47.1 dolů" )
      wire#w1
      S_Coil( "Klapka P47.1 dolů" )
   END_RUNG
   RUNG wire#w1
      R_Coil( "Klapka P47.1 nahoru" )
   END_RUNG
   // the same network as SCL:
   IF NOT "Globální řízení_DB".Automat AND #"Klapka P47.1 dolů" THEN
       "Klapka P47.1 dolů" := TRUE;
       "Klapka P47.1 nahoru" := FALSE;
   END_IF;
END_REGION

REGION Network 27
   RUNG wire#powerrail
      I_Contact( "Globální řízení_DB".Automat )
      Contact( "OPPovely".Linka1."P47.2 Start" )
      wire#w1
      Coil( "P 47.2 Start" )
   END_RUNG
   RUNG wire#powerrail
      Contact( "Globální řízení_DB".Automat )
      wire#w2
      I_Contact( "Karton na konci P47.2" )
   END_RUNG wire#w1
   RUNG wire#w2
      I_Contact( #"Karton na počítání" )
      I_Contact( #PlnáŘadaD49 )
   END_RUNG wire#w1
   // the same network as SCL:
   "P 47.2 Start" := (NOT "Globální řízení_DB".Automat AND "OPPovely".Linka1."P47.2 Start") OR ("Globální řízení_DB".Automat AND (NOT "Karton na konci P47.2" OR (NOT #"Karton na počítání" AND NOT #PlnáŘadaD49)));
END_REGION

REGION Network 28
   RUNG wire#powerrail
      Contact( "OPPovely Positivní Hrana".Linka1."Klapka P47.2" )
      wire#w1
      I_Contact( "Klapka 47.2 nahoru" )
      Coil( #"Klapka P47.2 nahoru" )
   END_RUNG
   RUNG wire#w1
      Contact( "Klapka 47.2 nahoru" )
      Coil( #"Klapka P47.2 dolů" )
   END_RUNG
   // the same network as SCL:
   #"Klapka P47.2 nahoru" := "OPPovely Positivní Hrana".Linka1."Klapka P47.2" AND NOT "Klapka 47.2 nahoru";
   #"Klapka P47.2 dolů" := "OPPovely Positivní Hrana".Linka1."Klapka P47.2" AND "Klapka 47.2 nahoru";
END_REGION

REGION Network 29
   RUNG wire#powerrail
      I_Contact( "Globální řízení_DB".Automat )
      Contact( #"Klapka P47.2 nahoru" )
      wire#w1
      S_Coil( "Klapka 47.2 nahoru" )
   END_RUNG
   RUNG wire#powerrail
      Contact( "Globální řízení_DB".Automat )
      Contact( #PlnáŘadaD49 )
      I_Contact( #"Karton na počítání" )
   END_RUNG wire#w1
   RUNG wire#w1
      R_Coil( "Klapka 47.2 dolů" )
   END_RUNG
   // the same network as SCL:
   IF (NOT "Globální řízení_DB".Automat AND #"Klapka P47.2 nahoru") OR ("Globální řízení_DB".Automat AND #PlnáŘadaD49 AND NOT #"Karton na počítání") THEN
       "Klapka 47.2 nahoru" := TRUE;
       "Klapka 47.2 dolů" := FALSE;
   END_IF;
END_REGION

REGION Network 30
   RUNG wire#powerrail
      I_Contact( "Globální řízení_DB".Automat )
      Contact( #"Klapka P47.2 dolů" )
      wire#w1
      S_Coil( "Klapka 47.2 dolů" )
   END_RUNG
   RUNG wire#powerrail
      Contact( "Globální řízení_DB".Automat )
      I_Contact( #PlnáŘadaD49 )
   END_RUNG wire#w1
   RUNG wire#w1
      R_Coil( "Klapka 47.2 nahoru" )
   END_RUNG
   // the same network as SCL:
   IF (NOT "Globální řízení_DB".Automat AND #"Klapka P47.2 dolů") OR ("Globální řízení_DB".Automat AND NOT #PlnáŘadaD49) THEN
       "Klapka 47.2 dolů" := TRUE;
       "Klapka 47.2 nahoru" := FALSE;
   END_IF;
END_REGION

REGION Network 31
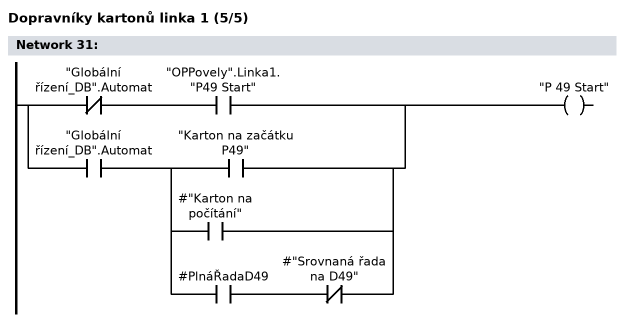
   RUNG wire#powerrail
      I_Contact( "Globální řízení_DB".Automat )
      Contact( "OPPovely".Linka1."P49 Start" )
      wire#w1
      Coil( "P 49 Start" )
   END_RUNG
   RUNG wire#powerrail
      Contact( "Globální řízení_DB".Automat )
      wire#w2
      Contact( "Karton na začátku P49" )
   END_RUNG wire#w1
   RUNG wire#w2
      Contact( #"Karton na počítání" )
   END_RUNG wire#w1
   RUNG wire#w2
      Contact( #PlnáŘadaD49 )
      I_Contact( #"Srovnaná řada na D49" )
   END_RUNG wire#w1
   // the same network as SCL:
   "P 49 Start" := (NOT "Globální řízení_DB".Automat AND "OPPovely".Linka1."P49 Start") OR ("Globální řízení_DB".Automat AND ("Karton na začátku P49" OR #"Karton na počítání" OR (#PlnáŘadaD49 AND NOT #"Srovnaná řada na D49")));
END_REGION
END_FUNCTION_BLOCK

FUNCTION_BLOCK "Globální řízení"   // FB6, LAD
{ S7_Optimized_Access := 'FALSE' }
VERSION : 0.1
   VAR
      Automat : Bool;
      "Automat Delay" : Bool;
      "Vyhodnocení hran_Instance" : "Vyhodnocení hran";
      "Vyhodnocení hran_Instance_Linka 1" : "Vyhodnocení hran";
   END_VAR
   VAR_TEMP
      Start : Bool;
      Stop : Bool;
   END_VAR
   VAR_TEMP   // added for the SCL form of the ladder/FBD networks
      _w1 : Bool;
      _s5time1 : S5Time;
   END_VAR
BEGIN

REGION Network 1
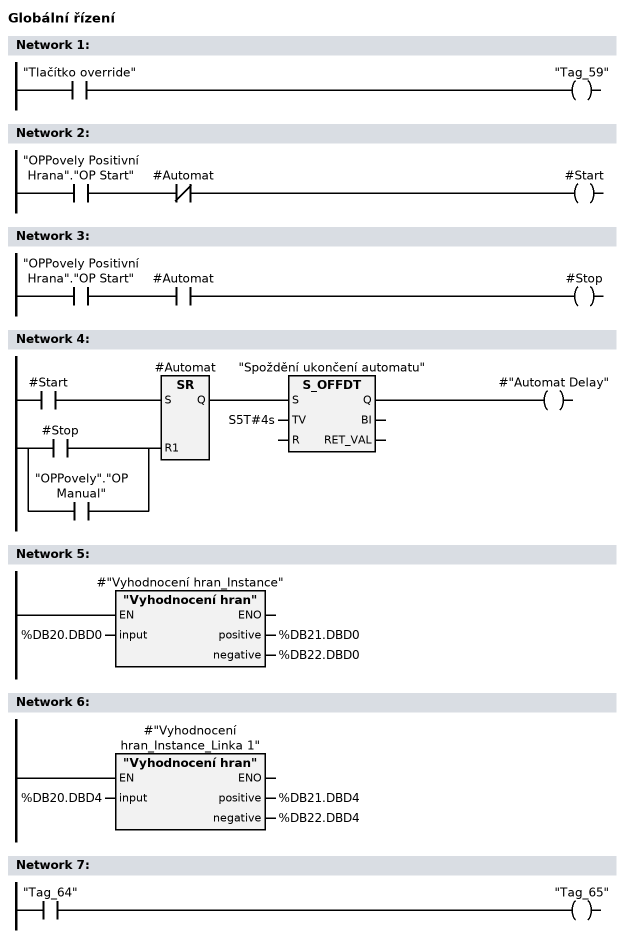
   RUNG wire#powerrail
      Contact( "Tlačítko override" )
      Coil( "Tag_59" )
   END_RUNG
   // the same network as SCL:
   "Tag_59" := "Tlačítko override";
END_REGION

REGION Network 2
   RUNG wire#powerrail
      Contact( "OPPovely Positivní Hrana"."OP Start" )
      I_Contact( #Automat )
      Coil( #Start )
   END_RUNG
   // the same network as SCL:
   #Start := "OPPovely Positivní Hrana"."OP Start" AND NOT #Automat;
END_REGION

REGION Network 3
   RUNG wire#powerrail
      Contact( "OPPovely Positivní Hrana"."OP Start" )
      Contact( #Automat )
      Coil( #Stop )
   END_RUNG
   // the same network as SCL:
   #Stop := "OPPovely Positivní Hrana"."OP Start" AND #Automat;
END_REGION

